gfCNCPoint5[28762] = {X 295.8044, Y 11.0396, Z -8.0000, A 0.000, B 0.000, C 0.000 }
gfCNCPoint5[28763] = {X 295.9180, Y 11.7127, Z -8.0000, A 0.000, B 0.000, C 0.000 }
gfCNCPoint5[28764] = {X 295.9354, Y 11.9495, Z -8.0000, A 0.000, B 0.000, C 0.000 }
gfCNCPoint5[28765] = {X 295.9411, Y 12.1868, Z -8.0000, A 0.000, B 0.000, C 0.000 }
gfCNCPoint5[28766] = {X 295.9409, Y 13.0237, Z -8.0000, A 0.000, B 0.000, C 0.000 }
gfCNCPoint5[28767] = {X 295.9342, Y 13.2382, Z -8.0000, A 0.000, B 0.000, C 0.000 }
gfCNCPoint5[28768] = {X 295.9180, Y 13.4521, Z -8.0000, A 0.000, B 0.000, C 0.000 }
gfCNCPoint5[28769] = {X 298.3067, Y 13.6853, Z -8.0000, A 0.000, B 0.000, C 0.000 }
gfCNCPoint5[28770] = {X 298.1362, Y 14.6931, Z -8.0000, A 0.000, B 0.000, C 0.000 }
gfCNCPoint5[28771] = {X 297.8263, Y 15.6671, Z -8.0000, A 0.000, B 0.000, C 0.000 }
gfCNCPoint5[28772] = {X 297.3830, Y 16.5881, Z -8.0000, A 0.000, B 0.000, C 0.000 }
gfCNCPoint5[28773] = {X 296.8150, Y 17.4380, Z -8.0000, A 0.000, B 0.000, C 0.000 }
gfCNCPoint5[28774] = {X 296.8153, Y 19.2365, Z -8.0000, A 0.000, B 0.000, C 0.000 }
gfCNCPoint5[28775] = {X 299.7981, Y 19.2365, Z -8.0000, A 0.000, B 0.000, C 0.000 }
gfCNCPoint5[28776] = {X 299.7982, Y 17.4377, Z -8.0000, A 0.000, B 0.000, C 0.000 }
gfCNCPoint5[28777] = {X 299.2303, Y 16.5879, Z -8.0000, A 0.000, B 0.000, C 0.000 }
gfCNCPoint5[28778] = {X 298.7871, Y 15.6670, Z -8.0000, A 0.000, B 0.000, C 0.000 }
gfCNCPoint5[28779] = {X 298.4771, Y 14.6930, Z -8.0000, A 0.000, B 0.000, C 0.000 }
gfCNCPoint5[28780] = {X 298.3067, Y 13.6853, Z -8.0000, A 0.000, B 0.000, C 0.000 }
gfCNCPoint5[28781] = {X 295.9180, Y 13.4521, Z -8.0000, A 0.000, B 0.000, C 0.000 }
gfCNCPoint5[28782] = {X 295.7561, Y 14.3091, Z -8.0000, A 0.000, B 0.000, C 0.000 }
gfCNCPoint5[28783] = {X 295.4442, Y 15.1235, Z -8.0000, A 0.000, B 0.000, C 0.000 }
gfCNCPoint5[28784] = {X 294.9923, Y 15.8694, Z -8.0000, A 0.000, B 0.000, C 0.000 }
gfCNCPoint5[28785] = {X 294.4149, Y 16.5230, Z -8.0000, A 0.000, B 0.000, C 0.000 }
gfCNCPoint5[28786] = {X 294.4149, Y 16.7686, Z -8.0000, A 0.000, B 0.000, C 0.000 }
gfCNCPoint5[28787] = {X 294.4156, Y 21.6365, Z -8.0000, A 0.000, B 0.000, C 0.000 }
gfCNCPoint5[28788] = {X 302.1980, Y 21.6365, Z -8.0000, A 0.000, B 0.000, C 0.000 }
gfCNCPoint5[28789] = {X 302.1982, Y 16.5227, Z -8.0000, A 0.000, B 0.000, C 0.000 }
gfCNCPoint5[28790] = {X 301.6209, Y 15.8692, Z -8.0000, A 0.000, B 0.000, C 0.000 }
gfCNCPoint5[28791] = {X 301.1691, Y 15.1233, Z -8.0000, A 0.000, B 0.000, C 0.000 }
gfCNCPoint5[28792] = {X 300.8573, Y 14.3090, Z -8.0000, A 0.000, B 0.000, C 0.000 }
gfCNCPoint5[28793] = {X 300.6953, Y 13.4521, Z -8.0000, A 0.000, B 0.000, C 0.000 }
gfCNCPoint5[28794] = {X 300.6791, Y 13.2371, Z -8.0000, A 0.000, B 0.000, C 0.000 }
gfCNCPoint5[28795] = {X 300.6724, Y 13.0215, Z -8.0000, A 0.000, B 0.000, C 0.000 }
gfCNCPoint5[28796] = {X 300.6723, Y 12.1868, Z -8.0000, A 0.000, B 0.000, C 0.000 }
gfCNCPoint5[28797] = {X 300.6780, Y 11.9495, Z -8.0000, A 0.000, B 0.000, C 0.000 }
gfCNCPoint5[28798] = {X 300.6953, Y 11.7127, Z -8.0000, A 0.000, B 0.000, C 0.000 }
gfCNCPoint5[28799] = {X 300.8090, Y 11.0396, Z -8.0000, A 0.000, B 0.000, C 0.000 }
gfCNCPoint5[28800] = {X 301.0155, Y 10.3890, Z -8.0000, A 0.000, B 0.000, C 0.000 }
gfCNCPoint5[28801] = {X 301.4602, Y 9.5279, Z -8.0000, A 0.000, B 0.000, C 0.000 }
gfCNCPoint5[28802] = {X 302.0663, Y 8.7718, Z -8.0000, A 0.000, B 0.000, C 0.000 }
gfCNCPoint5[28803] = {X 302.8099, Y 8.1502, Z -8.0000, A 0.000, B 0.000, C 0.000 }
gfCNCPoint5[28804] = {X 303.6616, Y 7.6879, Z -8.0000, A 0.000, B 0.000, C 0.000 }
gfCNCPoint5[28805] = {X 304.5879, Y 7.4030, Z -8.0000, A 0.000, B 0.000, C 0.000 }
gfCNCPoint5[28806] = {X 305.5523, Y 7.3068, Z -8.0000, A 0.000, B 0.000, C 0.000 }
gfCNCPoint5[28807] = {X 311.9957, Y 7.3068, Z -8.0000, A 0.000, B 0.000, C 0.000 }
gfCNCPoint5[28808] = {X 312.9478, Y 7.4006, Z -8.0000, A 0.000, B 0.000, C 0.000 }
gfCNCPoint5[28809] = {X 313.8632, Y 7.6783, Z -8.0000, A 0.000, B 0.000, C 0.000 }
gfCNCPoint5[28810] = {X 314.7069, Y 8.1292, Z -8.0000, A 0.000, B 0.000, C 0.000 }
gfCNCPoint5[28811] = {X 315.4464, Y 8.7361, Z -8.0000, A 0.000, B 0.000, C 0.000 }
gfCNCPoint5[28812] = {X 316.0533, Y 9.4756, Z -8.0000, A 0.000, B 0.000, C 0.000 }
gfCNCPoint5[28813] = {X 316.5043, Y 10.3193, Z -8.0000, A 0.000, B 0.000, C 0.000 }
gfCNCPoint5[28814] = {X 316.7820, Y 11.2348, Z -8.0000, A 0.000, B 0.000, C 0.000 }
gfCNCPoint5[28815] = {X 316.8757, Y 12.1868, Z -8.0000, A 0.000, B 0.000, C 0.000 }
gfCNCPoint5[28816] = {X 316.8755, Y 13.0237, Z -8.0000, A 0.000, B 0.000, C 0.000 }
gfCNCPoint5[28817] = {X 316.7682, Y 13.9967, Z -8.0000, A 0.000, B 0.000, C 0.000 }
gfCNCPoint5[28818] = {X 316.4689, Y 14.9287, Z -8.0000, A 0.000, B 0.000, C 0.000 }
gfCNCPoint5[28819] = {X 315.9896, Y 15.7823, Z -8.0000, A 0.000, B 0.000, C 0.000 }
gfCNCPoint5[28820] = {X 315.3495, Y 16.5229, Z -8.0000, A 0.000, B 0.000, C 0.000 }
gfCNCPoint5[28821] = {X 315.3493, Y 40.6637, Z -8.0000, A 0.000, B 0.000, C 0.000 }
gfCNCPoint5[28822] = {X 315.9899, Y 41.4051, Z -8.0000, A 0.000, B 0.000, C 0.000 }
gfCNCPoint5[28823] = {X 316.4695, Y 42.2595, Z -8.0000, A 0.000, B 0.000, C 0.000 }
gfCNCPoint5[28824] = {X 316.7687, Y 43.1925, Z -8.0000, A 0.000, B 0.000, C 0.000 }
gfCNCPoint5[28825] = {X 316.8755, Y 44.1664, Z -8.0000, A 0.000, B 0.000, C 0.000 }
gfCNCPoint5[28826] = {X 316.8757, Y 45.0000, Z -8.0000, A 0.000, B 0.000, C 0.000 }
gfCNCPoint5[28827] = {X 316.8749, Y 45.0899, Z -8.0000, A 0.000, B 0.000, C 0.000 }
gfCNCPoint5[28828] = {X 316.8724, Y 45.1799, Z -8.0000, A 0.000, B 0.000, C 0.000 }
gfCNCPoint5[28829] = {X 316.8594, Y 45.3987, Z -8.0000, A 0.000, B 0.000, C 0.000 }
gfCNCPoint5[28830] = {X 316.8366, Y 45.6167, Z -8.0000, A 0.000, B 0.000, C 0.000 }
gfCNCPoint5[28831] = {X 316.6062, Y 46.5992, Z -8.0000, A 0.000, B 0.000, C 0.000 }
gfCNCPoint5[28832] = {X 316.1787, Y 47.5134, Z -8.0000, A 0.000, B 0.000, C 0.000 }
gfCNCPoint5[28833] = {X 315.5723, Y 48.3200, Z -8.0000, A 0.000, B 0.000, C 0.000 }
gfCNCPoint5[28834] = {X 315.2205, Y 47.9934, Z -8.0000, A 0.000, B 0.000, C 0.000 }
gfCNCPoint5[28835] = {X 314.5413, Y 48.5889, Z -8.0000, A 0.000, B 0.000, C 0.000 }
gfCNCPoint5[28836] = {X 313.7548, Y 49.0331, Z -8.0000, A 0.000, B 0.000, C 0.000 }
gfCNCPoint5[28837] = {X 312.8942, Y 49.3073, Z -8.0000, A 0.000, B 0.000, C 0.000 }
gfCNCPoint5[28838] = {X 311.9957, Y 49.4000, Z -8.0000, A 0.000, B 0.000, C 0.000 }
gfCNCPoint5[28839] = {X 305.5523, Y 49.4000, Z -8.0000, A 0.000, B 0.000, C 0.000 }
gfCNCPoint5[28840] = {X 304.5732, Y 49.2897, Z -8.0000, A 0.000, B 0.000, C 0.000 }
gfCNCPoint5[28841] = {X 303.6432, Y 48.9643, Z -8.0000, A 0.000, B 0.000, C 0.000 }
gfCNCPoint5[28842] = {X 302.8089, Y 48.4401, Z -8.0000, A 0.000, B 0.000, C 0.000 }
gfCNCPoint5[28843] = {X 302.1122, Y 47.7433, Z -8.0000, A 0.000, B 0.000, C 0.000 }
gfCNCPoint5[28844] = {X 301.5880, Y 46.9091, Z -8.0000, A 0.000, B 0.000, C 0.000 }
gfCNCPoint5[28845] = {X 301.2626, Y 45.9791, Z -8.0000, A 0.000, B 0.000, C 0.000 }
gfCNCPoint5[28846] = {X 301.1523, Y 45.0000, Z -8.0000, A 0.000, B 0.000, C 0.000 }
gfCNCPoint5[28847] = {X 301.1524, Y 44.1996, Z -8.0000, A 0.000, B 0.000, C 0.000 }
gfCNCPoint5[28848] = {X 301.2693, Y 43.2561, Z -8.0000, A 0.000, B 0.000, C 0.000 }
gfCNCPoint5[28849] = {X 301.5719, Y 42.3548, Z -8.0000, A 0.000, B 0.000, C 0.000 }
gfCNCPoint5[28850] = {X 302.0480, Y 41.5318, Z -8.0000, A 0.000, B 0.000, C 0.000 }
gfCNCPoint5[28851] = {X 302.6784, Y 40.8201, Z -8.0000, A 0.000, B 0.000, C 0.000 }
gfCNCPoint5[28852] = {X 302.6784, Y 34.1143, Z -8.0000, A 0.000, B 0.000, C 0.000 }
gfCNCPoint5[28853] = {X 293.9354, Y 34.1143, Z -8.0000, A 0.000, B 0.000, C 0.000 }
gfCNCPoint5[28854] = {X 293.9349, Y 40.8654, Z -8.0000, A 0.000, B 0.000, C 0.000 }
gfCNCPoint5[28855] = {X 294.5750, Y 41.5604, Z -8.0000, A 0.000, B 0.000, C 0.000 }
gfCNCPoint5[28856] = {X 295.0555, Y 42.3739, Z -8.0000, A 0.000, B 0.000, C 0.000 }
gfCNCPoint5[28857] = {X 295.3554, Y 43.2699, Z -8.0000, A 0.000, B 0.000, C 0.000 }
gfCNCPoint5[28858] = {X 295.4611, Y 44.2088, Z -8.0000, A 0.000, B 0.000, C 0.000 }
gfCNCPoint5[28859] = {X 295.4611, Y 45.0000, Z -8.0000, A 0.000, B 0.000, C 0.000 }
gfCNCPoint5[28860] = {X 295.3508, Y 45.9791, Z -8.0000, A 0.000, B 0.000, C 0.000 }
gfCNCPoint5[28861] = {X 295.0254, Y 46.9091, Z -8.0000, A 0.000, B 0.000, C 0.000 }
gfCNCPoint5[28862] = {X 294.5012, Y 47.7434, Z -8.0000, A 0.000, B 0.000, C 0.000 }
gfCNCPoint5[28863] = {X 293.8045, Y 48.4401, Z -8.0000, A 0.000, B 0.000, C 0.000 }
gfCNCPoint5[28864] = {X 292.9702, Y 48.9643, Z -8.0000, A 0.000, B 0.000, C 0.000 }
gfCNCPoint5[28865] = {X 292.0402, Y 49.2897, Z -8.0000, A 0.000, B 0.000, C 0.000 }
gfCNCPoint5[28866] = {X 291.0611, Y 49.4000, Z -8.0000, A 0.000, B 0.000, C 0.000 }
gfCNCPoint5[28867] = {X 284.6177, Y 49.4000, Z -8.0000, A 0.000, B 0.000, C 0.000 }
gfCNCPoint5[28868] = {X 283.6386, Y 49.2897, Z -8.0000, A 0.000, B 0.000, C 0.000 }
gfCNCPoint5[28869] = {X 282.7086, Y 48.9643, Z -8.0000, A 0.000, B 0.000, C 0.000 }
gfCNCPoint5[28870] = {X 281.8743, Y 48.4401, Z -8.0000, A 0.000, B 0.000, C 0.000 }
gfCNCPoint5[28871] = {X 281.1776, Y 47.7433, Z -8.0000, A 0.000, B 0.000, C 0.000 }
gfCNCPoint5[28872] = {X 280.6534, Y 46.9091, Z -8.0000, A 0.000, B 0.000, C 0.000 }
gfCNCPoint5[28873] = {X 280.3280, Y 45.9791, Z -8.0000, A 0.000, B 0.000, C 0.000 }
gfCNCPoint5[28874] = {X 280.2177, Y 45.0000, Z -8.0000, A 0.000, B 0.000, C 0.000 }
gfCNCPoint5[28875] = {X 280.2177, Y 44.2072, Z -8.0000, A 0.000, B 0.000, C 0.000 }
gfCNCPoint5[28876] = {X 280.3216, Y 43.2699, Z -8.0000, A 0.000, B 0.000, C 0.000 }
gfCNCPoint5[28877] = {X 280.6210, Y 42.3756, Z -8.0000, A 0.000, B 0.000, C 0.000 }
gfCNCPoint5[28878] = {X 281.1024, Y 41.5647, Z -8.0000, A 0.000, B 0.000, C 0.000 }
gfCNCPoint5[28879] = {X 281.7441, Y 40.8737, Z -8.0000, A 0.000, B 0.000, C 0.000 }
gfCNCPoint5[28880] = {X 281.7443, Y 16.3102, Z -8.0000, A 0.000, B 0.000, C 0.000 }
gfCNCPoint5[28881] = {X 281.1000, Y 15.6212, Z -8.0000, A 0.000, B 0.000, C 0.000 }
gfCNCPoint5[28882] = {X 280.6175, Y 14.8106, Z -8.0000, A 0.000, B 0.000, C 0.000 }
gfCNCPoint5[28883] = {X 280.3188, Y 13.9159, Z -8.0000, A 0.000, B 0.000, C 0.000 }
gfCNCPoint5[28884] = {X 280.2177, Y 12.9780, Z -8.0000, A 0.000, B 0.000, C 0.000 }
gfCNCPoint5[28885] = {X 280.2177, Y 12.1868, Z -8.0000, A 0.000, B 0.000, C 0.000 }
gfCNCPoint5[28886] = {X 280.3280, Y 11.2077, Z -8.0000, A 0.000, B 0.000, C 0.000 }
gfCNCPoint5[28887] = {X 280.6534, Y 10.2777, Z -8.0000, A 0.000, B 0.000, C 0.000 }
gfCNCPoint5[28888] = {X 281.1776, Y 9.4435, Z -8.0000, A 0.000, B 0.000, C 0.000 }
gfCNCPoint5[28889] = {X 281.8743, Y 8.7468, Z -8.0000, A 0.000, B 0.000, C 0.000 }
gfCNCPoint5[28890] = {X 282.7086, Y 8.2226, Z -8.0000, A 0.000, B 0.000, C 0.000 }
gfCNCPoint5[28891] = {X 283.6386, Y 7.8971, Z -8.0000, A 0.000, B 0.000, C 0.000 }
gfCNCPoint5[28892] = {X 284.6177, Y 7.7868, Z -8.0000, A 0.000, B 0.000, C 0.000 }
gfCNCPoint5[28893] = {X 291.0611, Y 7.7868, Z -8.0000, A 0.000, B 0.000, C 0.000 }
gfCNCPoint5[28894] = {X 292.0402, Y 7.8971, Z -8.0000, A 0.000, B 0.000, C 0.000 }
gfCNCPoint5[28895] = {X 292.9702, Y 8.2226, Z -8.0000, A 0.000, B 0.000, C 0.000 }
gfCNCPoint5[28896] = {X 293.8045, Y 8.7468, Z -8.0000, A 0.000, B 0.000, C 0.000 }
gfCNCPoint5[28897] = {X 294.5012, Y 9.4435, Z -8.0000, A 0.000, B 0.000, C 0.000 }
gfCNCPoint5[28898] = {X 295.0254, Y 10.2777, Z -8.0000, A 0.000, B 0.000, C 0.000 }
gfCNCPoint5[28899] = {X 295.3508, Y 11.2077, Z -8.0000, A 0.000, B 0.000, C 0.000 }
gfCNCPoint5[28900] = {X 295.4611, Y 12.1868, Z -8.0000, A 0.000, B 0.000, C 0.000 }
gfCNCPoint5[28901] = {X 295.4609, Y 13.0233, Z -8.0000, A 0.000, B 0.000, C 0.000 }
gfCNCPoint5[28902] = {X 295.3527, Y 13.9490, Z -8.0000, A 0.000, B 0.000, C 0.000 }
gfCNCPoint5[28903] = {X 295.0519, Y 14.8311, Z -8.0000, A 0.000, B 0.000, C 0.000 }
gfCNCPoint5[28904] = {X 294.5721, Y 15.6300, Z -8.0000, A 0.000, B 0.000, C 0.000 }
gfCNCPoint5[28905] = {X 293.9348, Y 16.3100, Z -8.0000, A 0.000, B 0.000, C 0.000 }
gfCNCPoint5[28906] = {X 293.9349, Y 16.7687, Z -8.0000, A 0.000, B 0.000, C 0.000 }
gfCNCPoint5[28907] = {X 293.9356, Y 22.1165, Z -8.0000, A 0.000, B 0.000, C 0.000 }
gfCNCPoint5[28908] = {X 302.6780, Y 22.1165, Z -8.0000, A 0.000, B 0.000, C 0.000 }
gfCNCPoint5[28909] = {X 302.6782, Y 16.3097, Z -8.0000, A 0.000, B 0.000, C 0.000 }
gfCNCPoint5[28910] = {X 302.0342, Y 15.6207, Z -8.0000, A 0.000, B 0.000, C 0.000 }
gfCNCPoint5[28911] = {X 301.5519, Y 14.8102, Z -8.0000, A 0.000, B 0.000, C 0.000 }
gfCNCPoint5[28912] = {X 301.2533, Y 13.9156, Z -8.0000, A 0.000, B 0.000, C 0.000 }
gfCNCPoint5[28913] = {X 301.1523, Y 12.9780, Z -8.0000, A 0.000, B 0.000, C 0.000 }
gfCNCPoint5[28914] = {X 301.1523, Y 12.1868, Z -8.0000, A 0.000, B 0.000, C 0.000 }
gfCNCPoint5[28915] = {X 301.2626, Y 11.2077, Z -8.0000, A 0.000, B 0.000, C 0.000 }
gfCNCPoint5[28916] = {X 301.5880, Y 10.2777, Z -8.0000, A 0.000, B 0.000, C 0.000 }
gfCNCPoint5[28917] = {X 302.1122, Y 9.4435, Z -8.0000, A 0.000, B 0.000, C 0.000 }
gfCNCPoint5[28918] = {X 302.8089, Y 8.7468, Z -8.0000, A 0.000, B 0.000, C 0.000 }
gfCNCPoint5[28919] = {X 303.6432, Y 8.2226, Z -8.0000, A 0.000, B 0.000, C 0.000 }
gfCNCPoint5[28920] = {X 304.5732, Y 7.8971, Z -8.0000, A 0.000, B 0.000, C 0.000 }
gfCNCPoint5[28921] = {X 305.5523, Y 7.7868, Z -8.0000, A 0.000, B 0.000, C 0.000 }
gfCNCPoint5[28922] = {X 311.9957, Y 7.7868, Z -8.0000, A 0.000, B 0.000, C 0.000 }
gfCNCPoint5[28923] = {X 312.9748, Y 7.8971, Z -8.0000, A 0.000, B 0.000, C 0.000 }
gfCNCPoint5[28924] = {X 313.9048, Y 8.2226, Z -8.0000, A 0.000, B 0.000, C 0.000 }
gfCNCPoint5[28925] = {X 314.7391, Y 8.7468, Z -8.0000, A 0.000, B 0.000, C 0.000 }
gfCNCPoint5[28926] = {X 315.4358, Y 9.4435, Z -8.0000, A 0.000, B 0.000, C 0.000 }
gfCNCPoint5[28927] = {X 315.9600, Y 10.2777, Z -8.0000, A 0.000, B 0.000, C 0.000 }
gfCNCPoint5[28928] = {X 316.2854, Y 11.2077, Z -8.0000, A 0.000, B 0.000, C 0.000 }
gfCNCPoint5[28929] = {X 316.3957, Y 12.1868, Z -8.0000, A 0.000, B 0.000, C 0.000 }
gfCNCPoint5[28930] = {X 316.3955, Y 13.0233, Z -8.0000, A 0.000, B 0.000, C 0.000 }
gfCNCPoint5[28931] = {X 316.2873, Y 13.9489, Z -8.0000, A 0.000, B 0.000, C 0.000 }
gfCNCPoint5[28932] = {X 315.9865, Y 14.8310, Z -8.0000, A 0.000, B 0.000, C 0.000 }
gfCNCPoint5[28933] = {X 315.5068, Y 15.6299, Z -8.0000, A 0.000, B 0.000, C 0.000 }
gfCNCPoint5[28934] = {X 314.8695, Y 16.3099, Z -8.0000, A 0.000, B 0.000, C 0.000 }
gfCNCPoint5[28935] = {X 314.8693, Y 40.8767, Z -8.0000, A 0.000, B 0.000, C 0.000 }
gfCNCPoint5[28936] = {X 315.5135, Y 41.5658, Z -8.0000, A 0.000, B 0.000, C 0.000 }
gfCNCPoint5[28937] = {X 315.9960, Y 42.3763, Z -8.0000, A 0.000, B 0.000, C 0.000 }
gfCNCPoint5[28938] = {X 316.2946, Y 43.2710, Z -8.0000, A 0.000, B 0.000, C 0.000 }
gfCNCPoint5[28939] = {X 316.3957, Y 44.2089, Z -8.0000, A 0.000, B 0.000, C 0.000 }
gfCNCPoint5[28940] = {X 316.3957, Y 45.0000, Z -8.0000, A 0.000, B 0.000, C 0.000 }
gfCNCPoint5[28941] = {X 316.3190, Y 45.8182, Z -8.0000, A 0.000, B 0.000, C 0.000 }
gfCNCPoint5[28942] = {X 316.0914, Y 46.6079, Z -8.0000, A 0.000, B 0.000, C 0.000 }
gfCNCPoint5[28943] = {X 315.7209, Y 47.3415, Z -8.0000, A 0.000, B 0.000, C 0.000 }
gfCNCPoint5[28944] = {X 315.2205, Y 47.9934, Z -8.0000, A 0.000, B 0.000, C 0.000 }
gfCNCPoint5[28945] = {X 315.5723, Y 48.3200, Z -8.0000, A 0.000, B 0.000, C 0.000 }
gfCNCPoint5[28946] = {X 324.3107, Y 48.3200, Z -8.0000, A 0.000, B 0.000, C 0.000 }
gfCNCPoint5[28947] = {X 325.5555, Y 48.4004, Z -8.0000, A 0.000, B 0.000, C 0.000 }
gfCNCPoint5[28948] = {X 326.7797, Y 48.6402, Z -8.0000, A 0.000, B 0.000, C 0.000 }
gfCNCPoint5[28949] = {X 325.5882, Y 48.0963, Z -8.0000, A 0.000, B 0.000, C 0.000 }
gfCNCPoint5[28950] = {X 324.4810, Y 47.3966, Z -8.0000, A 0.000, B 0.000, C 0.000 }
gfCNCPoint5[28951] = {X 323.4784, Y 46.5538, Z -8.0000, A 0.000, B 0.000, C 0.000 }
gfCNCPoint5[28952] = {X 322.8382, Y 45.9295, Z -8.0000, A 0.000, B 0.000, C 0.000 }
gfCNCPoint5[28953] = {X 322.2180, Y 45.2650, Z -8.0000, A 0.000, B 0.000, C 0.000 }
gfCNCPoint5[28954] = {X 321.6628, Y 44.5452, Z -8.0000, A 0.000, B 0.000, C 0.000 }
gfCNCPoint5[28955] = {X 323.6300, Y 43.1703, Z -8.0000, A 0.000, B 0.000, C 0.000 }
gfCNCPoint5[28956] = {X 323.0063, Y 42.0918, Z -8.0000, A 0.000, B 0.000, C 0.000 }
gfCNCPoint5[28957] = {X 322.5757, Y 40.9227, Z -8.0000, A 0.000, B 0.000, C 0.000 }
gfCNCPoint5[28958] = {X 322.3506, Y 39.6973, Z -8.0000, A 0.000, B 0.000, C 0.000 }
gfCNCPoint5[28959] = {X 322.3379, Y 38.4514, Z -8.0000, A 0.000, B 0.000, C 0.000 }
gfCNCPoint5[28960] = {X 322.5377, Y 37.2217, Z -8.0000, A 0.000, B 0.000, C 0.000 }
gfCNCPoint5[28961] = {X 322.9443, Y 36.0440, Z -8.0000, A 0.000, B 0.000, C 0.000 }
gfCNCPoint5[28962] = {X 323.5458, Y 34.9529, Z -8.0000, A 0.000, B 0.000, C 0.000 }
gfCNCPoint5[28963] = {X 327.7840, Y 28.6158, Z -8.0000, A 0.000, B 0.000, C 0.000 }
gfCNCPoint5[28964] = {X 328.5200, Y 27.6906, Z -8.0000, A 0.000, B 0.000, C 0.000 }
gfCNCPoint5[28965] = {X 329.3960, Y 26.8968, Z -8.0000, A 0.000, B 0.000, C 0.000 }
gfCNCPoint5[28966] = {X 330.3889, Y 26.2552, Z -8.0000, A 0.000, B 0.000, C 0.000 }
gfCNCPoint5[28967] = {X 331.5063, Y 25.7713, Z -8.0000, A 0.000, B 0.000, C 0.000 }
gfCNCPoint5[28968] = {X 332.6887, Y 25.4804, Z -8.0000, A 0.000, B 0.000, C 0.000 }
gfCNCPoint5[28969] = {X 333.9031, Y 25.3907, Z -8.0000, A 0.000, B 0.000, C 0.000 }
gfCNCPoint5[28970] = {X 335.1154, Y 25.5046, Z -8.0000, A 0.000, B 0.000, C 0.000 }
gfCNCPoint5[28971] = {X 336.2918, Y 25.8191, Z -8.0000, A 0.000, B 0.000, C 0.000 }
gfCNCPoint5[28972] = {X 337.3993, Y 26.3252, Z -8.0000, A 0.000, B 0.000, C 0.000 }
gfCNCPoint5[28973] = {X 338.1754, Y 26.8291, Z -8.0000, A 0.000, B 0.000, C 0.000 }
gfCNCPoint5[28974] = {X 338.8812, Y 27.4274, Z -8.0000, A 0.000, B 0.000, C 0.000 }
gfCNCPoint5[28975] = {X 339.5028, Y 28.0267, Z -8.0000, A 0.000, B 0.000, C 0.000 }
gfCNCPoint5[28976] = {X 340.3317, Y 28.9981, Z -8.0000, A 0.000, B 0.000, C 0.000 }
gfCNCPoint5[28977] = {X 340.9781, Y 30.0993, Z -8.0000, A 0.000, B 0.000, C 0.000 }
gfCNCPoint5[28978] = {X 341.4222, Y 31.2965, Z -8.0000, A 0.000, B 0.000, C 0.000 }
gfCNCPoint5[28979] = {X 341.6502, Y 32.5529, Z -8.0000, A 0.000, B 0.000, C 0.000 }
gfCNCPoint5[28980] = {X 342.6387, Y 33.2799, Z -8.0000, A 0.000, B 0.000, C 0.000 }
gfCNCPoint5[28981] = {X 343.7299, Y 33.8413, Z -8.0000, A 0.000, B 0.000, C 0.000 }
gfCNCPoint5[28982] = {X 344.8962, Y 34.2227, Z -8.0000, A 0.000, B 0.000, C 0.000 }
gfCNCPoint5[28983] = {X 346.1081, Y 34.4147, Z -8.0000, A 0.000, B 0.000, C 0.000 }
gfCNCPoint5[28984] = {X 347.3352, Y 34.4123, Z -8.0000, A 0.000, B 0.000, C 0.000 }
gfCNCPoint5[28985] = {X 348.3044, Y 34.2866, Z -8.0000, A 0.000, B 0.000, C 0.000 }
gfCNCPoint5[28986] = {X 349.2397, Y 34.0036, Z -8.0000, A 0.000, B 0.000, C 0.000 }
gfCNCPoint5[28987] = {X 350.1160, Y 33.5708, Z -8.0000, A 0.000, B 0.000, C 0.000 }
gfCNCPoint5[28988] = {X 350.9093, Y 33.0001, Z -8.0000, A 0.000, B 0.000, C 0.000 }
gfCNCPoint5[28989] = {X 351.7850, Y 32.1491, Z -8.0000, A 0.000, B 0.000, C 0.000 }
gfCNCPoint5[28990] = {X 352.5431, Y 31.1918, Z -8.0000, A 0.000, B 0.000, C 0.000 }
gfCNCPoint5[28991] = {X 353.1707, Y 30.1444, Z -8.0000, A 0.000, B 0.000, C 0.000 }
gfCNCPoint5[28992] = {X 353.6573, Y 29.0244, Z -8.0000, A 0.000, B 0.000, C 0.000 }
gfCNCPoint5[28993] = {X 353.9945, Y 27.8508, Z -8.0000, A 0.000, B 0.000, C 0.000 }
gfCNCPoint5[28994] = {X 354.2220, Y 26.4400, Z -8.0000, A 0.000, B 0.000, C 0.000 }
gfCNCPoint5[28995] = {X 354.3140, Y 25.0140, Z -8.0000, A 0.000, B 0.000, C 0.000 }
gfCNCPoint5[28996] = {X 354.2698, Y 23.5857, Z -8.0000, A 0.000, B 0.000, C 0.000 }
gfCNCPoint5[28997] = {X 354.0897, Y 22.1681, Z -8.0000, A 0.000, B 0.000, C 0.000 }
gfCNCPoint5[28998] = {X 353.8250, Y 21.0254, Z -8.0000, A 0.000, B 0.000, C 0.000 }
gfCNCPoint5[28999] = {X 353.4119, Y 19.9275, Z -8.0000, A 0.000, B 0.000, C 0.000 }
gfCNCPoint5[29000] = {X 352.8576, Y 18.8937, Z -8.0000, A 0.000, B 0.000, C 0.000 }
gfCNCPoint5[29001] = {X 352.1718, Y 17.9421, Z -8.0000, A 0.000, B 0.000, C 0.000 }
gfCNCPoint5[29002] = {X 351.4219, Y 17.1690, Z -8.0000, A 0.000, B 0.000, C 0.000 }
gfCNCPoint5[29003] = {X 350.5492, Y 16.5376, Z -8.0000, A 0.000, B 0.000, C 0.000 }
gfCNCPoint5[29004] = {X 349.5804, Y 16.0671, Z -8.0000, A 0.000, B 0.000, C 0.000 }
gfCNCPoint5[29005] = {X 348.5446, Y 15.7717, Z -8.0000, A 0.000, B 0.000, C 0.000 }
gfCNCPoint5[29006] = {X 347.1584, Y 15.5996, Z -8.0000, A 0.000, B 0.000, C 0.000 }
gfCNCPoint5[29007] = {X 345.7616, Y 15.6148, Z -8.0000, A 0.000, B 0.000, C 0.000 }
gfCNCPoint5[29008] = {X 344.3794, Y 15.8170, Z -8.0000, A 0.000, B 0.000, C 0.000 }
gfCNCPoint5[29009] = {X 343.0368, Y 16.2026, Z -8.0000, A 0.000, B 0.000, C 0.000 }
gfCNCPoint5[29010] = {X 341.7580, Y 16.7646, Z -8.0000, A 0.000, B 0.000, C 0.000 }
gfCNCPoint5[29011] = {X 341.4304, Y 17.8590, Z -8.0000, A 0.000, B 0.000, C 0.000 }
gfCNCPoint5[29012] = {X 340.9357, Y 18.8888, Z -8.0000, A 0.000, B 0.000, C 0.000 }
gfCNCPoint5[29013] = {X 340.2859, Y 19.8284, Z -8.0000, A 0.000, B 0.000, C 0.000 }
gfCNCPoint5[29014] = {X 345.8684, Y 24.3755, Z -8.0000, A 0.000, B 0.000, C 0.000 }
gfCNCPoint5[29015] = {X 346.4660, Y 25.2106, Z -8.0000, A 0.000, B 0.000, C 0.000 }
gfCNCPoint5[29016] = {X 347.0029, Y 26.0860, Z -8.0000, A 0.000, B 0.000, C 0.000 }
gfCNCPoint5[29017] = {X 347.1049, Y 25.1804, Z -8.0000, A 0.000, B 0.000, C 0.000 }
gfCNCPoint5[29018] = {X 347.1005, Y 24.2691, Z -8.0000, A 0.000, B 0.000, C 0.000 }
gfCNCPoint5[29019] = {X 346.9895, Y 23.3646, Z -8.0000, A 0.000, B 0.000, C 0.000 }
gfCNCPoint5[29020] = {X 346.9483, Y 23.1618, Z -8.0000, A 0.000, B 0.000, C 0.000 }
gfCNCPoint5[29021] = {X 346.8824, Y 22.9657, Z -8.0000, A 0.000, B 0.000, C 0.000 }
gfCNCPoint5[29022] = {X 346.3965, Y 23.6858, Z -8.0000, A 0.000, B 0.000, C 0.000 }
gfCNCPoint5[29023] = {X 345.8684, Y 24.3755, Z -8.0000, A 0.000, B 0.000, C 0.000 }
gfCNCPoint5[29024] = {X 344.0076, Y 22.8598, Z -8.0000, A 0.000, B 0.000, C 0.000 }
gfCNCPoint5[29025] = {X 343.3277, Y 23.6257, Z -8.0000, A 0.000, B 0.000, C 0.000 }
gfCNCPoint5[29026] = {X 342.5854, Y 24.3313, Z -8.0000, A 0.000, B 0.000, C 0.000 }
gfCNCPoint5[29027] = {X 343.4620, Y 25.2275, Z -8.0000, A 0.000, B 0.000, C 0.000 }
gfCNCPoint5[29028] = {X 344.2409, Y 26.2098, Z -8.0000, A 0.000, B 0.000, C 0.000 }
gfCNCPoint5[29029] = {X 344.9138, Y 27.2675, Z -8.0000, A 0.000, B 0.000, C 0.000 }
gfCNCPoint5[29030] = {X 345.4656, Y 28.3710, Z -8.0000, A 0.000, B 0.000, C 0.000 }
gfCNCPoint5[29031] = {X 345.9019, Y 29.5251, Z -8.0000, A 0.000, B 0.000, C 0.000 }
gfCNCPoint5[29032] = {X 346.4628, Y 29.6282, Z -8.0000, A 0.000, B 0.000, C 0.000 }
gfCNCPoint5[29033] = {X 347.0330, Y 29.6206, Z -8.0000, A 0.000, B 0.000, C 0.000 }
gfCNCPoint5[29034] = {X 347.4389, Y 29.5545, Z -8.0000, A 0.000, B 0.000, C 0.000 }
gfCNCPoint5[29035] = {X 347.7946, Y 29.3479, Z -8.0000, A 0.000, B 0.000, C 0.000 }
gfCNCPoint5[29036] = {X 348.4743, Y 28.6286, Z -8.0000, A 0.000, B 0.000, C 0.000 }
gfCNCPoint5[29037] = {X 348.9844, Y 27.7806, Z -8.0000, A 0.000, B 0.000, C 0.000 }
gfCNCPoint5[29038] = {X 349.3014, Y 26.8431, Z -8.0000, A 0.000, B 0.000, C 0.000 }
gfCNCPoint5[29039] = {X 349.3362, Y 26.6688, Z -8.0000, A 0.000, B 0.000, C 0.000 }
gfCNCPoint5[29040] = {X 349.3680, Y 26.4938, Z -8.0000, A 0.000, B 0.000, C 0.000 }
gfCNCPoint5[29041] = {X 349.5008, Y 25.3209, Z -8.0000, A 0.000, B 0.000, C 0.000 }
gfCNCPoint5[29042] = {X 349.4971, Y 24.1405, Z -8.0000, A 0.000, B 0.000, C 0.000 }
gfCNCPoint5[29043] = {X 349.3568, Y 22.9684, Z -8.0000, A 0.000, B 0.000, C 0.000 }
gfCNCPoint5[29044] = {X 349.1791, Y 22.2566, Z -8.0000, A 0.000, B 0.000, C 0.000 }
gfCNCPoint5[29045] = {X 348.8767, Y 21.5882, Z -8.0000, A 0.000, B 0.000, C 0.000 }
gfCNCPoint5[29046] = {X 348.4593, Y 20.9848, Z -8.0000, A 0.000, B 0.000, C 0.000 }
gfCNCPoint5[29047] = {X 348.0918, Y 20.6609, Z -8.0000, A 0.000, B 0.000, C 0.000 }
gfCNCPoint5[29048] = {X 347.6348, Y 20.4847, Z -8.0000, A 0.000, B 0.000, C 0.000 }
gfCNCPoint5[29049] = {X 346.5774, Y 20.3831, Z -8.0000, A 0.000, B 0.000, C 0.000 }
gfCNCPoint5[29050] = {X 345.5199, Y 20.4829, Z -8.0000, A 0.000, B 0.000, C 0.000 }
gfCNCPoint5[29051] = {X 344.8333, Y 21.7156, Z -8.0000, A 0.000, B 0.000, C 0.000 }
gfCNCPoint5[29052] = {X 344.0076, Y 22.8598, Z -8.0000, A 0.000, B 0.000, C 0.000 }
gfCNCPoint5[29053] = {X 342.1467, Y 21.3441, Z -8.0000, A 0.000, B 0.000, C 0.000 }
gfCNCPoint5[29054] = {X 341.6020, Y 21.9578, Z -8.0000, A 0.000, B 0.000, C 0.000 }
gfCNCPoint5[29055] = {X 341.0072, Y 22.5232, Z -8.0000, A 0.000, B 0.000, C 0.000 }
gfCNCPoint5[29056] = {X 340.7216, Y 22.7630, Z -8.0000, A 0.000, B 0.000, C 0.000 }
gfCNCPoint5[29057] = {X 340.4270, Y 22.9916, Z -8.0000, A 0.000, B 0.000, C 0.000 }
gfCNCPoint5[29058] = {X 339.6616, Y 23.5549, Z -8.0000, A 0.000, B 0.000, C 0.000 }
gfCNCPoint5[29059] = {X 339.1300, Y 23.9121, Z -8.0000, A 0.000, B 0.000, C 0.000 }
gfCNCPoint5[29060] = {X 338.5759, Y 24.2333, Z -8.0000, A 0.000, B 0.000, C 0.000 }
gfCNCPoint5[29061] = {X 339.6077, Y 24.9034, Z -8.0000, A 0.000, B 0.000, C 0.000 }
gfCNCPoint5[29062] = {X 340.5463, Y 25.6990, Z -8.0000, A 0.000, B 0.000, C 0.000 }
gfCNCPoint5[29063] = {X 341.1848, Y 26.3147, Z -8.0000, A 0.000, B 0.000, C 0.000 }
gfCNCPoint5[29064] = {X 342.1205, Y 27.3794, Z -8.0000, A 0.000, B 0.000, C 0.000 }
gfCNCPoint5[29065] = {X 342.8906, Y 28.5694, Z -8.0000, A 0.000, B 0.000, C 0.000 }
gfCNCPoint5[29066] = {X 343.4787, Y 29.8590, Z -8.0000, A 0.000, B 0.000, C 0.000 }
gfCNCPoint5[29067] = {X 343.8721, Y 31.2207, Z -8.0000, A 0.000, B 0.000, C 0.000 }
gfCNCPoint5[29068] = {X 344.6396, Y 31.6203, Z -8.0000, A 0.000, B 0.000, C 0.000 }
gfCNCPoint5[29069] = {X 345.4616, Y 31.8904, Z -8.0000, A 0.000, B 0.000, C 0.000 }
gfCNCPoint5[29070] = {X 346.3165, Y 32.0237, Z -8.0000, A 0.000, B 0.000, C 0.000 }
gfCNCPoint5[29071] = {X 347.1817, Y 32.0168, Z -8.0000, A 0.000, B 0.000, C 0.000 }
gfCNCPoint5[29072] = {X 347.9625, Y 31.9015, Z -8.0000, A 0.000, B 0.000, C 0.000 }
gfCNCPoint5[29073] = {X 348.6981, Y 31.6158, Z -8.0000, A 0.000, B 0.000, C 0.000 }
gfCNCPoint5[29074] = {X 349.3520, Y 31.1739, Z -8.0000, A 0.000, B 0.000, C 0.000 }
gfCNCPoint5[29075] = {X 350.1526, Y 30.3706, Z -8.0000, A 0.000, B 0.000, C 0.000 }
gfCNCPoint5[29076] = {X 350.8130, Y 29.4485, Z -8.0000, A 0.000, B 0.000, C 0.000 }
gfCNCPoint5[29077] = {X 351.3158, Y 28.4318, Z -8.0000, A 0.000, B 0.000, C 0.000 }
gfCNCPoint5[29078] = {X 351.6479, Y 27.3474, Z -8.0000, A 0.000, B 0.000, C 0.000 }
gfCNCPoint5[29079] = {X 351.8764, Y 25.7621, Z -8.0000, A 0.000, B 0.000, C 0.000 }
gfCNCPoint5[29080] = {X 351.9017, Y 24.1606, Z -8.0000, A 0.000, B 0.000, C 0.000 }
gfCNCPoint5[29081] = {X 351.7234, Y 22.5689, Z -8.0000, A 0.000, B 0.000, C 0.000 }
gfCNCPoint5[29082] = {X 351.4415, Y 21.4556, Z -8.0000, A 0.000, B 0.000, C 0.000 }
gfCNCPoint5[29083] = {X 350.9674, Y 20.4097, Z -8.0000, A 0.000, B 0.000, C 0.000 }
gfCNCPoint5[29084] = {X 350.3159, Y 19.4639, Z -8.0000, A 0.000, B 0.000, C 0.000 }
gfCNCPoint5[29085] = {X 349.6854, Y 18.8481, Z -8.0000, A 0.000, B 0.000, C 0.000 }
gfCNCPoint5[29086] = {X 348.9297, Y 18.3948, Z -8.0000, A 0.000, B 0.000, C 0.000 }
gfCNCPoint5[29087] = {X 348.0897, Y 18.1282, Z -8.0000, A 0.000, B 0.000, C 0.000 }
gfCNCPoint5[29088] = {X 346.9971, Y 17.9943, Z -8.0000, A 0.000, B 0.000, C 0.000 }
gfCNCPoint5[29089] = {X 345.8964, Y 18.0117, Z -8.0000, A 0.000, B 0.000, C 0.000 }
gfCNCPoint5[29090] = {X 344.8086, Y 18.1800, Z -8.0000, A 0.000, B 0.000, C 0.000 }
gfCNCPoint5[29091] = {X 343.7541, Y 18.4960, Z -8.0000, A 0.000, B 0.000, C 0.000 }
gfCNCPoint5[29092] = {X 343.3271, Y 19.5041, Z -8.0000, A 0.000, B 0.000, C 0.000 }
gfCNCPoint5[29093] = {X 342.7890, Y 20.4575, Z -8.0000, A 0.000, B 0.000, C 0.000 }
gfCNCPoint5[29094] = {X 342.1467, Y 21.3441, Z -8.0000, A 0.000, B 0.000, C 0.000 }
gfCNCPoint5[29095] = {X 340.2859, Y 19.8284, Z -8.0000, A 0.000, B 0.000, C 0.000 }
gfCNCPoint5[29096] = {X 339.6798, Y 20.4856, Z -8.0000, A 0.000, B 0.000, C 0.000 }
gfCNCPoint5[29097] = {X 338.9976, Y 21.0636, Z -8.0000, A 0.000, B 0.000, C 0.000 }
gfCNCPoint5[29098] = {X 338.2497, Y 21.6140, Z -8.0000, A 0.000, B 0.000, C 0.000 }
gfCNCPoint5[29099] = {X 337.8538, Y 21.8795, Z -8.0000, A 0.000, B 0.000, C 0.000 }
gfCNCPoint5[29100] = {X 337.4413, Y 22.1185, Z -8.0000, A 0.000, B 0.000, C 0.000 }
gfCNCPoint5[29101] = {X 336.3239, Y 22.6023, Z -8.0000, A 0.000, B 0.000, C 0.000 }
gfCNCPoint5[29102] = {X 335.1415, Y 22.8932, Z -8.0000, A 0.000, B 0.000, C 0.000 }
gfCNCPoint5[29103] = {X 333.9271, Y 22.9829, Z -8.0000, A 0.000, B 0.000, C 0.000 }
gfCNCPoint5[29104] = {X 332.7148, Y 22.8690, Z -8.0000, A 0.000, B 0.000, C 0.000 }
gfCNCPoint5[29105] = {X 331.5384, Y 22.5546, Z -8.0000, A 0.000, B 0.000, C 0.000 }
gfCNCPoint5[29106] = {X 330.4309, Y 22.0485, Z -8.0000, A 0.000, B 0.000, C 0.000 }
gfCNCPoint5[29107] = {X 329.5144, Y 21.4374, Z -8.0000, A 0.000, B 0.000, C 0.000 }
gfCNCPoint5[29108] = {X 328.7005, Y 20.6950, Z -8.0000, A 0.000, B 0.000, C 0.000 }
gfCNCPoint5[29109] = {X 328.0081, Y 19.8382, Z -8.0000, A 0.000, B 0.000, C 0.000 }
gfCNCPoint5[29110] = {X 327.4528, Y 18.8869, Z -8.0000, A 0.000, B 0.000, C 0.000 }
gfCNCPoint5[29111] = {X 323.9321, Y 11.6443, Z -8.0000, A 0.000, B 0.000, C 0.000 }
gfCNCPoint5[29112] = {X 323.5337, Y 10.6421, Z -8.0000, A 0.000, B 0.000, C 0.000 }
gfCNCPoint5[29113] = {X 323.2878, Y 9.5921, Z -8.0000, A 0.000, B 0.000, C 0.000 }
gfCNCPoint5[29114] = {X 323.1997, Y 8.5173, Z -8.0000, A 0.000, B 0.000, C 0.000 }
gfCNCPoint5[29115] = {X 323.2713, Y 7.4412, Z -8.0000, A 0.000, B 0.000, C 0.000 }
gfCNCPoint5[29116] = {X 323.4720, Y 6.4883, Z -8.0000, A 0.000, B 0.000, C 0.000 }
gfCNCPoint5[29117] = {X 323.7980, Y 5.5707, Z -8.0000, A 0.000, B 0.000, C 0.000 }
gfCNCPoint5[29118] = {X 324.2436, Y 4.7048, Z -8.0000, A 0.000, B 0.000, C 0.000 }
gfCNCPoint5[29119] = {X 168.0207, Y 4.7048, Z -8.0000, A 0.000, B 0.000, C 0.000 }
gfCNCPoint5[29120] = {X 168.0207, Y 9.5048, Z -8.0000, A 0.000, B 0.000, C 0.000 }
gfCNCPoint5[29121] = {X 166.5360, Y 9.5048, Z -8.0000, A 0.000, B 0.000, C 0.000 }
gfCNCPoint5[29122] = {X 166.5855, Y 9.9931, Z -8.0000, A 0.000, B 0.000, C 0.000 }
gfCNCPoint5[29123] = {X 166.6021, Y 10.4835, Z -8.0000, A 0.000, B 0.000, C 0.000 }
gfCNCPoint5[29124] = {X 166.6021, Y 13.0969, Z -8.0000, A 0.000, B 0.000, C 0.000 }
gfCNCPoint5[29125] = {X 166.8569, Y 11.8209, Z -8.0000, A 0.000, B 0.000, C 0.000 }
gfCNCPoint5[29126] = {X 167.3349, Y 10.6107, Z -8.0000, A 0.000, B 0.000, C 0.000 }
gfCNCPoint5[29127] = {X 168.0207, Y 9.5048, Z -8.0000, A 0.000, B 0.000, C 0.000 }
gfCNCPoint5[29128] = {X 168.0207, Y 7.1048, Z -8.0000, A 0.000, B 0.000, C 0.000 }
gfCNCPoint5[29129] = {X 162.8433, Y 7.1048, Z -8.0000, A 0.000, B 0.000, C 0.000 }
gfCNCPoint5[29130] = {X 163.4702, Y 7.9130, Z -8.0000, A 0.000, B 0.000, C 0.000 }
gfCNCPoint5[29131] = {X 163.9148, Y 8.8340, Z -8.0000, A 0.000, B 0.000, C 0.000 }
gfCNCPoint5[29132] = {X 164.1578, Y 9.8275, Z -8.0000, A 0.000, B 0.000, C 0.000 }
gfCNCPoint5[29133] = {X 164.1910, Y 10.1547, Z -8.0000, A 0.000, B 0.000, C 0.000 }
gfCNCPoint5[29134] = {X 164.2021, Y 10.4835, Z -8.0000, A 0.000, B 0.000, C 0.000 }
gfCNCPoint5[29135] = {X 164.2021, Y 17.4615, Z -8.0000, A 0.000, B 0.000, C 0.000 }
gfCNCPoint5[29136] = {X 164.1140, Y 18.3847, Z -8.0000, A 0.000, B 0.000, C 0.000 }
gfCNCPoint5[29137] = {X 163.8528, Y 19.2746, Z -8.0000, A 0.000, B 0.000, C 0.000 }
gfCNCPoint5[29138] = {X 163.4280, Y 20.0990, Z -8.0000, A 0.000, B 0.000, C 0.000 }
gfCNCPoint5[29139] = {X 162.8549, Y 20.8281, Z -8.0000, A 0.000, B 0.000, C 0.000 }
gfCNCPoint5[29140] = {X 162.1542, Y 21.4357, Z -8.0000, A 0.000, B 0.000, C 0.000 }
gfCNCPoint5[29141] = {X 161.3512, Y 21.8997, Z -8.0000, A 0.000, B 0.000, C 0.000 }
gfCNCPoint5[29142] = {X 160.4749, Y 22.2034, Z -8.0000, A 0.000, B 0.000, C 0.000 }
gfCNCPoint5[29143] = {X 162.1759, Y 29.1996, Z -8.0000, A 0.000, B 0.000, C 0.000 }
gfCNCPoint5[29144] = {X 161.1136, Y 29.4080, Z -8.0000, A 0.000, B 0.000, C 0.000 }
gfCNCPoint5[29145] = {X 160.0370, Y 29.5204, Z -8.0000, A 0.000, B 0.000, C 0.000 }
gfCNCPoint5[29146] = {X 160.0366, Y 38.3362, Z -8.0000, A 0.000, B 0.000, C 0.000 }
gfCNCPoint5[29147] = {X 160.6847, Y 39.6934, Z -8.0000, A 0.000, B 0.000, C 0.000 }
gfCNCPoint5[29148] = {X 161.1595, Y 41.1206, Z -8.0000, A 0.000, B 0.000, C 0.000 }
gfCNCPoint5[29149] = {X 162.0518, Y 41.1205, Z -8.0000, A 0.000, B 0.000, C 0.000 }
gfCNCPoint5[29150] = {X 161.8695, Y 40.3467, Z -8.0000, A 0.000, B 0.000, C 0.000 }
gfCNCPoint5[29151] = {X 161.7169, Y 39.5666, Z -8.0000, A 0.000, B 0.000, C 0.000 }
gfCNCPoint5[29152] = {X 161.5938, Y 38.7932, Z -8.0000, A 0.000, B 0.000, C 0.000 }
gfCNCPoint5[29153] = {X 161.3791, Y 36.8687, Z -8.0000, A 0.000, B 0.000, C 0.000 }
gfCNCPoint5[29154] = {X 161.3302, Y 34.9328, Z -8.0000, A 0.000, B 0.000, C 0.000 }
gfCNCPoint5[29155] = {X 161.4475, Y 32.9999, Z -8.0000, A 0.000, B 0.000, C 0.000 }
gfCNCPoint5[29156] = {X 161.7301, Y 31.0841, Z -8.0000, A 0.000, B 0.000, C 0.000 }
gfCNCPoint5[29157] = {X 162.1759, Y 29.1996, Z -8.0000, A 0.000, B 0.000, C 0.000 }
gfCNCPoint5[29158] = {X 161.6089, Y 26.8675, Z -8.0000, A 0.000, B 0.000, C 0.000 }
gfCNCPoint5[29159] = {X 160.4737, Y 27.0728, Z -8.0000, A 0.000, B 0.000, C 0.000 }
gfCNCPoint5[29160] = {X 159.3221, Y 27.1415, Z -8.0000, A 0.000, B 0.000, C 0.000 }
gfCNCPoint5[29161] = {X 158.6622, Y 27.1415, Z -8.0000, A 0.000, B 0.000, C 0.000 }
gfCNCPoint5[29162] = {X 158.1489, Y 27.1263, Z -8.0000, A 0.000, B 0.000, C 0.000 }
gfCNCPoint5[29163] = {X 157.6371, Y 27.0839, Z -8.0000, A 0.000, B 0.000, C 0.000 }
gfCNCPoint5[29164] = {X 157.6365, Y 38.9958, Z -8.0000, A 0.000, B 0.000, C 0.000 }
gfCNCPoint5[29165] = {X 158.2204, Y 40.0482, Z -8.0000, A 0.000, B 0.000, C 0.000 }
gfCNCPoint5[29166] = {X 158.6695, Y 41.1647, Z -8.0000, A 0.000, B 0.000, C 0.000 }
gfCNCPoint5[29167] = {X 158.9769, Y 42.3282, Z -8.0000, A 0.000, B 0.000, C 0.000 }
gfCNCPoint5[29168] = {X 159.1379, Y 43.5209, Z -8.0000, A 0.000, B 0.000, C 0.000 }
gfCNCPoint5[29169] = {X 165.4258, Y 43.5200, Z -8.0000, A 0.000, B 0.000, C 0.000 }
gfCNCPoint5[29170] = {X 164.8366, Y 42.0454, Z -8.0000, A 0.000, B 0.000, C 0.000 }
gfCNCPoint5[29171] = {X 164.3769, Y 40.5255, Z -8.0000, A 0.000, B 0.000, C 0.000 }
gfCNCPoint5[29172] = {X 164.2176, Y 39.8500, Z -8.0000, A 0.000, B 0.000, C 0.000 }
gfCNCPoint5[29173] = {X 164.0838, Y 39.1689, Z -8.0000, A 0.000, B 0.000, C 0.000 }
gfCNCPoint5[29174] = {X 163.9647, Y 38.4207, Z -8.0000, A 0.000, B 0.000, C 0.000 }
gfCNCPoint5[29175] = {X 163.7485, Y 36.2699, Z -8.0000, A 0.000, B 0.000, C 0.000 }
gfCNCPoint5[29176] = {X 163.7638, Y 34.1082, Z -8.0000, A 0.000, B 0.000, C 0.000 }
gfCNCPoint5[29177] = {X 164.0104, Y 31.9607, Z -8.0000, A 0.000, B 0.000, C 0.000 }
gfCNCPoint5[29178] = {X 164.4855, Y 29.8518, Z -8.0000, A 0.000, B 0.000, C 0.000 }
gfCNCPoint5[29179] = {X 164.8364, Y 28.7346, Z -8.0000, A 0.000, B 0.000, C 0.000 }
gfCNCPoint5[29180] = {X 165.2515, Y 27.6396, Z -8.0000, A 0.000, B 0.000, C 0.000 }
gfCNCPoint5[29181] = {X 165.8682, Y 26.3072, Z -8.0000, A 0.000, B 0.000, C 0.000 }
gfCNCPoint5[29182] = {X 166.6029, Y 25.0360, Z -8.0000, A 0.000, B 0.000, C 0.000 }
gfCNCPoint5[29183] = {X 167.4497, Y 23.8365, Z -8.0000, A 0.000, B 0.000, C 0.000 }
gfCNCPoint5[29184] = {X 167.1640, Y 23.1367, Z -8.0000, A 0.000, B 0.000, C 0.000 }
gfCNCPoint5[29185] = {X 166.2875, Y 24.1836, Z -8.0000, A 0.000, B 0.000, C 0.000 }
gfCNCPoint5[29186] = {X 165.2724, Y 25.0968, Z -8.0000, A 0.000, B 0.000, C 0.000 }
gfCNCPoint5[29187] = {X 164.1389, Y 25.8580, Z -8.0000, A 0.000, B 0.000, C 0.000 }
gfCNCPoint5[29188] = {X 162.9096, Y 26.4522, Z -8.0000, A 0.000, B 0.000, C 0.000 }
gfCNCPoint5[29189] = {X 161.6089, Y 26.8675, Z -8.0000, A 0.000, B 0.000, C 0.000 }
gfCNCPoint5[29190] = {X 161.0419, Y 24.5355, Z -8.0000, A 0.000, B 0.000, C 0.000 }
gfCNCPoint5[29191] = {X 160.1882, Y 24.6898, Z -8.0000, A 0.000, B 0.000, C 0.000 }
gfCNCPoint5[29192] = {X 159.3221, Y 24.7415, Z -8.0000, A 0.000, B 0.000, C 0.000 }
gfCNCPoint5[29193] = {X 158.6699, Y 24.7415, Z -8.0000, A 0.000, B 0.000, C 0.000 }
gfCNCPoint5[29194] = {X 158.2835, Y 24.7301, Z -8.0000, A 0.000, B 0.000, C 0.000 }
gfCNCPoint5[29195] = {X 157.8982, Y 24.6982, Z -8.0000, A 0.000, B 0.000, C 0.000 }
gfCNCPoint5[29196] = {X 156.9783, Y 24.5375, Z -8.0000, A 0.000, B 0.000, C 0.000 }
gfCNCPoint5[29197] = {X 156.0865, Y 24.2609, Z -8.0000, A 0.000, B 0.000, C 0.000 }
gfCNCPoint5[29198] = {X 155.2372, Y 23.8728, Z -8.0000, A 0.000, B 0.000, C 0.000 }
gfCNCPoint5[29199] = {X 155.2365, Y 39.7518, Z -8.0000, A 0.000, B 0.000, C 0.000 }
gfCNCPoint5[29200] = {X 155.8272, Y 40.6433, Z -8.0000, A 0.000, B 0.000, C 0.000 }
gfCNCPoint5[29201] = {X 156.2813, Y 41.6115, Z -8.0000, A 0.000, B 0.000, C 0.000 }
gfCNCPoint5[29202] = {X 156.5892, Y 42.6357, Z -8.0000, A 0.000, B 0.000, C 0.000 }
gfCNCPoint5[29203] = {X 156.7441, Y 43.6938, Z -8.0000, A 0.000, B 0.000, C 0.000 }
gfCNCPoint5[29204] = {X 156.7580, Y 43.9467, Z -8.0000, A 0.000, B 0.000, C 0.000 }
gfCNCPoint5[29205] = {X 156.7631, Y 44.1999, Z -8.0000, A 0.000, B 0.000, C 0.000 }
gfCNCPoint5[29206] = {X 156.7628, Y 45.0700, Z -8.0000, A 0.000, B 0.000, C 0.000 }
gfCNCPoint5[29207] = {X 156.7347, Y 45.6426, Z -8.0000, A 0.000, B 0.000, C 0.000 }
gfCNCPoint5[29208] = {X 156.6616, Y 46.2112, Z -8.0000, A 0.000, B 0.000, C 0.000 }
gfCNCPoint5[29209] = {X 157.9054, Y 46.0005, Z -8.0000, A 0.000, B 0.000, C 0.000 }
gfCNCPoint5[29210] = {X 159.1644, Y 45.9207, Z -8.0000, A 0.000, B 0.000, C 0.000 }
gfCNCPoint5[29211] = {X 159.2312, Y 45.9202, Z -8.0000, A 0.000, B 0.000, C 0.000 }
gfCNCPoint5[29212] = {X 159.2980, Y 45.9200, Z -8.0000, A 0.000, B 0.000, C 0.000 }
gfCNCPoint5[29213] = {X 169.6787, Y 45.9200, Z -8.0000, A 0.000, B 0.000, C 0.000 }
gfCNCPoint5[29214] = {X 168.8976, Y 44.8498, Z -8.0000, A 0.000, B 0.000, C 0.000 }
gfCNCPoint5[29215] = {X 168.2078, Y 43.7186, Z -8.0000, A 0.000, B 0.000, C 0.000 }
gfCNCPoint5[29216] = {X 167.6139, Y 42.5342, Z -8.0000, A 0.000, B 0.000, C 0.000 }
gfCNCPoint5[29217] = {X 167.1231, Y 41.3128, Z -8.0000, A 0.000, B 0.000, C 0.000 }
gfCNCPoint5[29218] = {X 166.7344, Y 40.0552, Z -8.0000, A 0.000, B 0.000, C 0.000 }
gfCNCPoint5[29219] = {X 166.4505, Y 38.7698, Z -8.0000, A 0.000, B 0.000, C 0.000 }
gfCNCPoint5[29220] = {X 166.3357, Y 38.0485, Z -8.0000, A 0.000, B 0.000, C 0.000 }
gfCNCPoint5[29221] = {X 166.1443, Y 36.1221, Z -8.0000, A 0.000, B 0.000, C 0.000 }
gfCNCPoint5[29222] = {X 166.1636, Y 34.1864, Z -8.0000, A 0.000, B 0.000, C 0.000 }
gfCNCPoint5[29223] = {X 166.3935, Y 32.2642, Z -8.0000, A 0.000, B 0.000, C 0.000 }
gfCNCPoint5[29224] = {X 166.8312, Y 30.3785, Z -8.0000, A 0.000, B 0.000, C 0.000 }
gfCNCPoint5[29225] = {X 167.4715, Y 28.5516, Z -8.0000, A 0.000, B 0.000, C 0.000 }
gfCNCPoint5[29226] = {X 168.2321, Y 26.9815, Z -8.0000, A 0.000, B 0.000, C 0.000 }
gfCNCPoint5[29227] = {X 169.1845, Y 25.5199, Z -8.0000, A 0.000, B 0.000, C 0.000 }
gfCNCPoint5[29228] = {X 170.3136, Y 24.1899, Z -8.0000, A 0.000, B 0.000, C 0.000 }
gfCNCPoint5[29229] = {X 169.9862, Y 23.6218, Z -8.0000, A 0.000, B 0.000, C 0.000 }
gfCNCPoint5[29230] = {X 169.7113, Y 23.0265, Z -8.0000, A 0.000, B 0.000, C 0.000 }
gfCNCPoint5[29231] = {X 167.1001, Y 16.6309, Z -8.0000, A 0.000, B 0.000, C 0.000 }
gfCNCPoint5[29232] = {X 166.7820, Y 15.6636, Z -8.0000, A 0.000, B 0.000, C 0.000 }
gfCNCPoint5[29233] = {X 166.6021, Y 14.6613, Z -8.0000, A 0.000, B 0.000, C 0.000 }
gfCNCPoint5[29234] = {X 166.6021, Y 17.4615, Z -8.0000, A 0.000, B 0.000, C 0.000 }
gfCNCPoint5[29235] = {X 166.5130, Y 18.5970, Z -8.0000, A 0.000, B 0.000, C 0.000 }
gfCNCPoint5[29236] = {X 166.2479, Y 19.7047, Z -8.0000, A 0.000, B 0.000, C 0.000 }
gfCNCPoint5[29237] = {X 165.8132, Y 20.7575, Z -8.0000, A 0.000, B 0.000, C 0.000 }
gfCNCPoint5[29238] = {X 165.2197, Y 21.7296, Z -8.0000, A 0.000, B 0.000, C 0.000 }
gfCNCPoint5[29239] = {X 164.3789, Y 22.6987, Z -8.0000, A 0.000, B 0.000, C 0.000 }
gfCNCPoint5[29240] = {X 163.3810, Y 23.5050, Z -8.0000, A 0.000, B 0.000, C 0.000 }
gfCNCPoint5[29241] = {X 162.2570, Y 24.1237, Z -8.0000, A 0.000, B 0.000, C 0.000 }
gfCNCPoint5[29242] = {X 161.0419, Y 24.5355, Z -8.0000, A 0.000, B 0.000, C 0.000 }
gfCNCPoint5[29243] = {X 160.4749, Y 22.2034, Z -8.0000, A 0.000, B 0.000, C 0.000 }
gfCNCPoint5[29244] = {X 159.9026, Y 22.3069, Z -8.0000, A 0.000, B 0.000, C 0.000 }
gfCNCPoint5[29245] = {X 159.3221, Y 22.3415, Z -8.0000, A 0.000, B 0.000, C 0.000 }
gfCNCPoint5[29246] = {X 158.6776, Y 22.3415, Z -8.0000, A 0.000, B 0.000, C 0.000 }
gfCNCPoint5[29247] = {X 157.8807, Y 22.2738, Z -8.0000, A 0.000, B 0.000, C 0.000 }
gfCNCPoint5[29248] = {X 157.1053, Y 22.0776, Z -8.0000, A 0.000, B 0.000, C 0.000 }
gfCNCPoint5[29249] = {X 156.3721, Y 21.7581, Z -8.0000, A 0.000, B 0.000, C 0.000 }
gfCNCPoint5[29250] = {X 155.5228, Y 21.1803, Z -8.0000, A 0.000, B 0.000, C 0.000 }
gfCNCPoint5[29251] = {X 154.8123, Y 20.4383, Z -8.0000, A 0.000, B 0.000, C 0.000 }
gfCNCPoint5[29252] = {X 152.8374, Y 20.4389, Z -8.0000, A 0.000, B 0.000, C 0.000 }
gfCNCPoint5[29253] = {X 152.8364, Y 40.6543, Z -8.0000, A 0.000, B 0.000, C 0.000 }
gfCNCPoint5[29254] = {X 153.1745, Y 41.0198, Z -8.0000, A 0.000, B 0.000, C 0.000 }
gfCNCPoint5[29255] = {X 153.6802, Y 41.7242, Z -8.0000, A 0.000, B 0.000, C 0.000 }
gfCNCPoint5[29256] = {X 154.0540, Y 42.5068, Z -8.0000, A 0.000, B 0.000, C 0.000 }
gfCNCPoint5[29257] = {X 154.2840, Y 43.3429, Z -8.0000, A 0.000, B 0.000, C 0.000 }
gfCNCPoint5[29258] = {X 154.3631, Y 44.2065, Z -8.0000, A 0.000, B 0.000, C 0.000 }
gfCNCPoint5[29259] = {X 154.3629, Y 45.0469, Z -8.0000, A 0.000, B 0.000, C 0.000 }
gfCNCPoint5[29260] = {X 154.3440, Y 45.4308, Z -8.0000, A 0.000, B 0.000, C 0.000 }
gfCNCPoint5[29261] = {X 154.2951, Y 45.8119, Z -8.0000, A 0.000, B 0.000, C 0.000 }
gfCNCPoint5[29262] = {X 154.0370, Y 46.7541, Z -8.0000, A 0.000, B 0.000, C 0.000 }
gfCNCPoint5[29263] = {X 153.5963, Y 47.6260, Z -8.0000, A 0.000, B 0.000, C 0.000 }
gfCNCPoint5[29264] = {X 152.9909, Y 48.3926, Z -8.0000, A 0.000, B 0.000, C 0.000 }
gfCNCPoint5[29265] = {X 152.2448, Y 49.0233, Z -8.0000, A 0.000, B 0.000, C 0.000 }
gfCNCPoint5[29266] = {X 151.3881, Y 49.4928, Z -8.0000, A 0.000, B 0.000, C 0.000 }
gfCNCPoint5[29267] = {X 150.4551, Y 49.7822, Z -8.0000, A 0.000, B 0.000, C 0.000 }
gfCNCPoint5[29268] = {X 149.4831, Y 49.8800, Z -8.0000, A 0.000, B 0.000, C 0.000 }
gfCNCPoint5[29269] = {X 143.0396, Y 49.8800, Z -8.0000, A 0.000, B 0.000, C 0.000 }
gfCNCPoint5[29270] = {X 142.0923, Y 49.7872, Z -8.0000, A 0.000, B 0.000, C 0.000 }
gfCNCPoint5[29271] = {X 141.1811, Y 49.5122, Z -8.0000, A 0.000, B 0.000, C 0.000 }
gfCNCPoint5[29272] = {X 140.3405, Y 49.0656, Z -8.0000, A 0.000, B 0.000, C 0.000 }
gfCNCPoint5[29273] = {X 139.6026, Y 48.4643, Z -8.0000, A 0.000, B 0.000, C 0.000 }
gfCNCPoint5[29274] = {X 138.9955, Y 47.7312, Z -8.0000, A 0.000, B 0.000, C 0.000 }
gfCNCPoint5[29275] = {X 138.5423, Y 46.8942, Z -8.0000, A 0.000, B 0.000, C 0.000 }
gfCNCPoint5[29276] = {X 138.2601, Y 45.9852, Z -8.0000, A 0.000, B 0.000, C 0.000 }
gfCNCPoint5[29277] = {X 138.1598, Y 45.0386, Z -8.0000, A 0.000, B 0.000, C 0.000 }
gfCNCPoint5[29278] = {X 138.1601, Y 44.1417, Z -8.0000, A 0.000, B 0.000, C 0.000 }
gfCNCPoint5[29279] = {X 138.2148, Y 43.4769, Z -8.0000, A 0.000, B 0.000, C 0.000 }
gfCNCPoint5[29280] = {X 138.3597, Y 42.8258, Z -8.0000, A 0.000, B 0.000, C 0.000 }
gfCNCPoint5[29281] = {X 129.1532, Y 40.1052, Z -8.0000, A 0.000, B 0.000, C 0.000 }
gfCNCPoint5[29282] = {X 129.5665, Y 38.9035, Z -8.0000, A 0.000, B 0.000, C 0.000 }
gfCNCPoint5[29283] = {X 130.0836, Y 37.7426, Z -8.0000, A 0.000, B 0.000, C 0.000 }
gfCNCPoint5[29284] = {X 130.0836, Y 31.6021, Z -8.0000, A 0.000, B 0.000, C 0.000 }
gfCNCPoint5[29285] = {X 129.2066, Y 31.3798, Z -8.0000, A 0.000, B 0.000, C 0.000 }
gfCNCPoint5[29286] = {X 128.3452, Y 31.1032, Z -8.0000, A 0.000, B 0.000, C 0.000 }
gfCNCPoint5[29287] = {X 128.3453, Y 38.3312, Z -8.0000, A 0.000, B 0.000, C 0.000 }
gfCNCPoint5[29288] = {X 128.7851, Y 39.2019, Z -8.0000, A 0.000, B 0.000, C 0.000 }
gfCNCPoint5[29289] = {X 129.1532, Y 40.1052, Z -8.0000, A 0.000, B 0.000, C 0.000 }
gfCNCPoint5[29290] = {X 131.4548, Y 40.7854, Z -8.0000, A 0.000, B 0.000, C 0.000 }
gfCNCPoint5[29291] = {X 131.9017, Y 39.5320, Z -8.0000, A 0.000, B 0.000, C 0.000 }
gfCNCPoint5[29292] = {X 132.4836, Y 38.3354, Z -8.0000, A 0.000, B 0.000, C 0.000 }
gfCNCPoint5[29293] = {X 132.4836, Y 29.5202, Z -8.0000, A 0.000, B 0.000, C 0.000 }
gfCNCPoint5[29294] = {X 131.3527, Y 29.3994, Z -8.0000, A 0.000, B 0.000, C 0.000 }
gfCNCPoint5[29295] = {X 130.2382, Y 29.1727, Z -8.0000, A 0.000, B 0.000, C 0.000 }
gfCNCPoint5[29296] = {X 129.1500, Y 28.8422, Z -8.0000, A 0.000, B 0.000, C 0.000 }
gfCNCPoint5[29297] = {X 128.0256, Y 28.3769, Z -8.0000, A 0.000, B 0.000, C 0.000 }
gfCNCPoint5[29298] = {X 126.9537, Y 27.8009, Z -8.0000, A 0.000, B 0.000, C 0.000 }
gfCNCPoint5[29299] = {X 125.9452, Y 27.1200, Z -8.0000, A 0.000, B 0.000, C 0.000 }
gfCNCPoint5[29300] = {X 125.9453, Y 38.9915, Z -8.0000, A 0.000, B 0.000, C 0.000 }
gfCNCPoint5[29301] = {X 126.4743, Y 39.9295, Z -8.0000, A 0.000, B 0.000, C 0.000 }
gfCNCPoint5[29302] = {X 126.8960, Y 40.9205, Z -8.0000, A 0.000, B 0.000, C 0.000 }
gfCNCPoint5[29303] = {X 127.2098, Y 41.9730, Z -8.0000, A 0.000, B 0.000, C 0.000 }
gfCNCPoint5[29304] = {X 127.4025, Y 43.0542, Z -8.0000, A 0.000, B 0.000, C 0.000 }
gfCNCPoint5[29305] = {X 127.4714, Y 44.1502, Z -8.0000, A 0.000, B 0.000, C 0.000 }
gfCNCPoint5[29306] = {X 127.4716, Y 45.0000, Z -8.0000, A 0.000, B 0.000, C 0.000 }
gfCNCPoint5[29307] = {X 127.4070, Y 46.1159, Z -8.0000, A 0.000, B 0.000, C 0.000 }
gfCNCPoint5[29308] = {X 127.2143, Y 47.2168, Z -8.0000, A 0.000, B 0.000, C 0.000 }
gfCNCPoint5[29309] = {X 126.8960, Y 48.2883, Z -8.0000, A 0.000, B 0.000, C 0.000 }
gfCNCPoint5[29310] = {X 126.2883, Y 49.6376, Z -8.0000, A 0.000, B 0.000, C 0.000 }
gfCNCPoint5[29311] = {X 125.4821, Y 50.8786, Z -8.0000, A 0.000, B 0.000, C 0.000 }
gfCNCPoint5[29312] = {X 124.4962, Y 51.9821, Z -8.0000, A 0.000, B 0.000, C 0.000 }
gfCNCPoint5[29313] = {X 123.3536, Y 52.9225, Z -8.0000, A 0.000, B 0.000, C 0.000 }
gfCNCPoint5[29314] = {X 122.0810, Y 53.6778, Z -8.0000, A 0.000, B 0.000, C 0.000 }
gfCNCPoint5[29315] = {X 120.7081, Y 54.2302, Z -8.0000, A 0.000, B 0.000, C 0.000 }
gfCNCPoint5[29316] = {X 119.2671, Y 54.5669, Z -8.0000, A 0.000, B 0.000, C 0.000 }
gfCNCPoint5[29317] = {X 117.7916, Y 54.6800, Z -8.0000, A 0.000, B 0.000, C 0.000 }
gfCNCPoint5[29318] = {X 111.9185, Y 54.6800, Z -8.0000, A 0.000, B 0.000, C 0.000 }
gfCNCPoint5[29319] = {X 111.7456, Y 54.6785, Z -8.0000, A 0.000, B 0.000, C 0.000 }
gfCNCPoint5[29320] = {X 111.5728, Y 54.6738, Z -8.0000, A 0.000, B 0.000, C 0.000 }
gfCNCPoint5[29321] = {X 111.0585, Y 69.0646, Z -8.0000, A 0.000, B 0.000, C 0.000 }
gfCNCPoint5[29322] = {X 109.0296, Y 68.9061, Z -8.0000, A 0.000, B 0.000, C 0.000 }
gfCNCPoint5[29323] = {X 107.0213, Y 68.5768, Z -8.0000, A 0.000, B 0.000, C 0.000 }
gfCNCPoint5[29324] = {X 105.0765, Y 68.8983, Z -8.0000, A 0.000, B 0.000, C 0.000 }
gfCNCPoint5[29325] = {X 103.1119, Y 69.0597, Z -8.0000, A 0.000, B 0.000, C 0.000 }
gfCNCPoint5[29326] = {X 101.1407, Y 69.0599, Z -8.0000, A 0.000, B 0.000, C 0.000 }
gfCNCPoint5[29327] = {X 99.1761, Y 68.8989, Z -8.0000, A 0.000, B 0.000, C 0.000 }
gfCNCPoint5[29328] = {X 97.2313, Y 68.5777, Z -8.0000, A 0.000, B 0.000, C 0.000 }
gfCNCPoint5[29329] = {X 95.6131, Y 68.8563, Z -8.0000, A 0.000, B 0.000, C 0.000 }
gfCNCPoint5[29330] = {X 93.9796, Y 69.0240, Z -8.0000, A 0.000, B 0.000, C 0.000 }
gfCNCPoint5[29331] = {X 92.3385, Y 69.0800, Z -8.0000, A 0.000, B 0.000, C 0.000 }
gfCNCPoint5[29332] = {X 86.6884, Y 69.0800, Z -8.0000, A 0.000, B 0.000, C 0.000 }
gfCNCPoint5[29333] = {X 84.7315, Y 70.2669, Z -8.0000, A 0.000, B 0.000, C 0.000 }
gfCNCPoint5[29334] = {X 82.6867, Y 71.2952, Z -8.0000, A 0.000, B 0.000, C 0.000 }
gfCNCPoint5[29335] = {X 107.2713, Y 71.2952, Z -8.0000, A 0.000, B 0.000, C 0.000 }
gfCNCPoint5[29336] = {X 109.1257, Y 70.1133, Z -8.0000, A 0.000, B 0.000, C 0.000 }
gfCNCPoint5[29337] = {X 111.0585, Y 69.0646, Z -8.0000, A 0.000, B 0.000, C 0.000 }
gfCNCPoint5[29338] = {X 111.1442, Y 66.6662, Z -8.0000, A 0.000, B 0.000, C 0.000 }
gfCNCPoint5[29339] = {X 109.0696, Y 66.4920, Z -8.0000, A 0.000, B 0.000, C 0.000 }
gfCNCPoint5[29340] = {X 107.0213, Y 66.1197, Z -8.0000, A 0.000, B 0.000, C 0.000 }
gfCNCPoint5[29341] = {X 105.0796, Y 66.4776, Z -8.0000, A 0.000, B 0.000, C 0.000 }
gfCNCPoint5[29342] = {X 103.1135, Y 66.6574, Z -8.0000, A 0.000, B 0.000, C 0.000 }
gfCNCPoint5[29343] = {X 101.1392, Y 66.6576, Z -8.0000, A 0.000, B 0.000, C 0.000 }
gfCNCPoint5[29344] = {X 99.1730, Y 66.4782, Z -8.0000, A 0.000, B 0.000, C 0.000 }
gfCNCPoint5[29345] = {X 97.2313, Y 66.1207, Z -8.0000, A 0.000, B 0.000, C 0.000 }
gfCNCPoint5[29346] = {X 95.6161, Y 66.4308, Z -8.0000, A 0.000, B 0.000, C 0.000 }
gfCNCPoint5[29347] = {X 93.9821, Y 66.6176, Z -8.0000, A 0.000, B 0.000, C 0.000 }
gfCNCPoint5[29348] = {X 92.3385, Y 66.6800, Z -8.0000, A 0.000, B 0.000, C 0.000 }
gfCNCPoint5[29349] = {X 85.9487, Y 66.6800, Z -8.0000, A 0.000, B 0.000, C 0.000 }
gfCNCPoint5[29350] = {X 83.8778, Y 67.9936, Z -8.0000, A 0.000, B 0.000, C 0.000 }
gfCNCPoint5[29351] = {X 81.6943, Y 69.1100, Z -8.0000, A 0.000, B 0.000, C 0.000 }
gfCNCPoint5[29352] = {X 79.6014, Y 69.9549, Z -8.0000, A 0.000, B 0.000, C 0.000 }
gfCNCPoint5[29353] = {X 77.4441, Y 70.6185, Z -8.0000, A 0.000, B 0.000, C 0.000 }
gfCNCPoint5[29354] = {X 75.2381, Y 71.0959, Z -8.0000, A 0.000, B 0.000, C 0.000 }
gfCNCPoint5[29355] = {X 72.9995, Y 71.3838, Z -8.0000, A 0.000, B 0.000, C 0.000 }
gfCNCPoint5[29356] = {X 70.7445, Y 71.4800, Z -8.0000, A 0.000, B 0.000, C 0.000 }
gfCNCPoint5[29357] = {X 64.1851, Y 71.4800, Z -8.0000, A 0.000, B 0.000, C 0.000 }
gfCNCPoint5[29358] = {X 62.0752, Y 71.3958, Z -8.0000, A 0.000, B 0.000, C 0.000 }
gfCNCPoint5[29359] = {X 59.9787, Y 71.1438, Z -8.0000, A 0.000, B 0.000, C 0.000 }
gfCNCPoint5[29360] = {X 57.9089, Y 70.7255, Z -8.0000, A 0.000, B 0.000, C 0.000 }
gfCNCPoint5[29361] = {X 55.8790, Y 70.1436, Z -8.0000, A 0.000, B 0.000, C 0.000 }
gfCNCPoint5[29362] = {X 53.8492, Y 70.7255, Z -8.0000, A 0.000, B 0.000, C 0.000 }
gfCNCPoint5[29363] = {X 51.7794, Y 71.1438, Z -8.0000, A 0.000, B 0.000, C 0.000 }
gfCNCPoint5[29364] = {X 49.6829, Y 71.3958, Z -8.0000, A 0.000, B 0.000, C 0.000 }
gfCNCPoint5[29365] = {X 47.5729, Y 71.4800, Z -8.0000, A 0.000, B 0.000, C 0.000 }
gfCNCPoint5[29366] = {X 40.6393, Y 71.4800, Z -8.0000, A 0.000, B 0.000, C 0.000 }
gfCNCPoint5[29367] = {X 38.8062, Y 71.4165, Z -8.0000, A 0.000, B 0.000, C 0.000 }
gfCNCPoint5[29368] = {X 36.9818, Y 71.2262, Z -8.0000, A 0.000, B 0.000, C 0.000 }
gfCNCPoint5[29369] = {X 34.3986, Y 72.0364, Z -8.0000, A 0.000, B 0.000, C 0.000 }
gfCNCPoint5[29370] = {X 31.7542, Y 72.6168, Z -8.0000, A 0.000, B 0.000, C 0.000 }
gfCNCPoint5[29371] = {X 30.3314, Y 73.1755, Z -8.0000, A 0.000, B 0.000, C 0.000 }
gfCNCPoint5[29372] = {X 28.8938, Y 73.6952, Z -8.0000, A 0.000, B 0.000, C 0.000 }
gfCNCPoint5[29373] = {X 108.0335, Y 73.6952, Z -8.0000, A 0.000, B 0.000, C 0.000 }
gfCNCPoint5[29374] = {X 110.0293, Y 72.3691, Z -8.0000, A 0.000, B 0.000, C 0.000 }
gfCNCPoint5[29375] = {X 112.1282, Y 71.2131, Z -8.0000, A 0.000, B 0.000, C 0.000 }
gfCNCPoint5[29376] = {X 113.1244, Y 70.7406, Z -8.0000, A 0.000, B 0.000, C 0.000 }
gfCNCPoint5[29377] = {X 114.1380, Y 70.3064, Z -8.0000, A 0.000, B 0.000, C 0.000 }
gfCNCPoint5[29378] = {X 117.4405, Y 66.6800, Z -8.0000, A 0.000, B 0.000, C 0.000 }
gfCNCPoint5[29379] = {X 111.9185, Y 66.6800, Z -8.0000, A 0.000, B 0.000, C 0.000 }
gfCNCPoint5[29380] = {X 111.5313, Y 66.6765, Z -8.0000, A 0.000, B 0.000, C 0.000 }
gfCNCPoint5[29381] = {X 111.1442, Y 66.6662, Z -8.0000, A 0.000, B 0.000, C 0.000 }
gfCNCPoint5[29382] = {X 111.2299, Y 64.2677, Z -8.0000, A 0.000, B 0.000, C 0.000 }
gfCNCPoint5[29383] = {X 109.1084, Y 64.0741, Z -8.0000, A 0.000, B 0.000, C 0.000 }
gfCNCPoint5[29384] = {X 107.0213, Y 63.6477, Z -8.0000, A 0.000, B 0.000, C 0.000 }
gfCNCPoint5[29385] = {X 105.0841, Y 64.0514, Z -8.0000, A 0.000, B 0.000, C 0.000 }
gfCNCPoint5[29386] = {X 103.1158, Y 64.2545, Z -8.0000, A 0.000, B 0.000, C 0.000 }
gfCNCPoint5[29387] = {X 101.1370, Y 64.2547, Z -8.0000, A 0.000, B 0.000, C 0.000 }
gfCNCPoint5[29388] = {X 99.1686, Y 64.0521, Z -8.0000, A 0.000, B 0.000, C 0.000 }
gfCNCPoint5[29389] = {X 97.2313, Y 63.6488, Z -8.0000, A 0.000, B 0.000, C 0.000 }
gfCNCPoint5[29390] = {X 95.6204, Y 63.9986, Z -8.0000, A 0.000, B 0.000, C 0.000 }
gfCNCPoint5[29391] = {X 93.9855, Y 64.2095, Z -8.0000, A 0.000, B 0.000, C 0.000 }
gfCNCPoint5[29392] = {X 92.3385, Y 64.2800, Z -8.0000, A 0.000, B 0.000, C 0.000 }
gfCNCPoint5[29393] = {X 85.8951, Y 64.2800, Z -8.0000, A 0.000, B 0.000, C 0.000 }
gfCNCPoint5[29394] = {X 85.5417, Y 64.2768, Z -8.0000, A 0.000, B 0.000, C 0.000 }
gfCNCPoint5[29395] = {X 85.1884, Y 64.2670, Z -8.0000, A 0.000, B 0.000, C 0.000 }
gfCNCPoint5[29396] = {X 83.3593, Y 65.5113, Z -8.0000, A 0.000, B 0.000, C 0.000 }
gfCNCPoint5[29397] = {X 81.4238, Y 66.5824, Z -8.0000, A 0.000, B 0.000, C 0.000 }
gfCNCPoint5[29398] = {X 79.3981, Y 67.4713, Z -8.0000, A 0.000, B 0.000, C 0.000 }
gfCNCPoint5[29399] = {X 77.2994, Y 68.1706, Z -8.0000, A 0.000, B 0.000, C 0.000 }
gfCNCPoint5[29400] = {X 75.1454, Y 68.6744, Z -8.0000, A 0.000, B 0.000, C 0.000 }
gfCNCPoint5[29401] = {X 72.9543, Y 68.9784, Z -8.0000, A 0.000, B 0.000, C 0.000 }
gfCNCPoint5[29402] = {X 70.7445, Y 69.0800, Z -8.0000, A 0.000, B 0.000, C 0.000 }
gfCNCPoint5[29403] = {X 64.1851, Y 69.0800, Z -8.0000, A 0.000, B 0.000, C 0.000 }
gfCNCPoint5[29404] = {X 62.0678, Y 68.9867, Z -8.0000, A 0.000, B 0.000, C 0.000 }
gfCNCPoint5[29405] = {X 59.9669, Y 68.7076, Z -8.0000, A 0.000, B 0.000, C 0.000 }
gfCNCPoint5[29406] = {X 57.8986, Y 68.2449, Z -8.0000, A 0.000, B 0.000, C 0.000 }
gfCNCPoint5[29407] = {X 55.8790, Y 67.6021, Z -8.0000, A 0.000, B 0.000, C 0.000 }
gfCNCPoint5[29408] = {X 53.8595, Y 68.2449, Z -8.0000, A 0.000, B 0.000, C 0.000 }
gfCNCPoint5[29409] = {X 51.7912, Y 68.7076, Z -8.0000, A 0.000, B 0.000, C 0.000 }
gfCNCPoint5[29410] = {X 49.6903, Y 68.9867, Z -8.0000, A 0.000, B 0.000, C 0.000 }
gfCNCPoint5[29411] = {X 47.5729, Y 69.0800, Z -8.0000, A 0.000, B 0.000, C 0.000 }
gfCNCPoint5[29412] = {X 40.6393, Y 69.0800, Z -8.0000, A 0.000, B 0.000, C 0.000 }
gfCNCPoint5[29413] = {X 38.6756, Y 68.9998, Z -8.0000, A 0.000, B 0.000, C 0.000 }
gfCNCPoint5[29414] = {X 36.7249, Y 68.7597, Z -8.0000, A 0.000, B 0.000, C 0.000 }
gfCNCPoint5[29415] = {X 34.8830, Y 69.4002, Z -8.0000, A 0.000, B 0.000, C 0.000 }
gfCNCPoint5[29416] = {X 33.0015, Y 69.9128, Z -8.0000, A 0.000, B 0.000, C 0.000 }
gfCNCPoint5[29417] = {X 31.0892, Y 70.2952, Z -8.0000, A 0.000, B 0.000, C 0.000 }
gfCNCPoint5[29418] = {X 29.6075, Y 70.8834, Z -8.0000, A 0.000, B 0.000, C 0.000 }
gfCNCPoint5[29419] = {X 28.1088, Y 71.4272, Z -8.0000, A 0.000, B 0.000, C 0.000 }
gfCNCPoint5[29420] = {X 27.6142, Y 71.5956, Z -8.0000, A 0.000, B 0.000, C 0.000 }
gfCNCPoint5[29421] = {X 27.1180, Y 71.7593, Z -8.0000, A 0.000, B 0.000, C 0.000 }
gfCNCPoint5[29422] = {X 25.5190, Y 72.2532, Z -8.0000, A 0.000, B 0.000, C 0.000 }
gfCNCPoint5[29423] = {X 23.9033, Y 72.6897, Z -8.0000, A 0.000, B 0.000, C 0.000 }
gfCNCPoint5[29424] = {X 23.9033, Y 76.0952, Z -8.0000, A 0.000, B 0.000, C 0.000 }
gfCNCPoint5[29425] = {X 108.8316, Y 76.0952, Z -8.0000, A 0.000, B 0.000, C 0.000 }
gfCNCPoint5[29426] = {X 110.4007, Y 74.9741, Z -8.0000, A 0.000, B 0.000, C 0.000 }
gfCNCPoint5[29427] = {X 112.0471, Y 73.9702, Z -8.0000, A 0.000, B 0.000, C 0.000 }
gfCNCPoint5[29428] = {X 113.7623, Y 73.0888, Z -8.0000, A 0.000, B 0.000, C 0.000 }
gfCNCPoint5[29429] = {X 115.5371, Y 72.3345, Z -8.0000, A 0.000, B 0.000, C 0.000 }
gfCNCPoint5[29430] = {X 123.7242, Y 63.3445, Z -8.0000, A 0.000, B 0.000, C 0.000 }
gfCNCPoint5[29431] = {X 121.7828, Y 63.8624, Z -8.0000, A 0.000, B 0.000, C 0.000 }
gfCNCPoint5[29432] = {X 119.7981, Y 64.1753, Z -8.0000, A 0.000, B 0.000, C 0.000 }
gfCNCPoint5[29433] = {X 117.7916, Y 64.2800, Z -8.0000, A 0.000, B 0.000, C 0.000 }
gfCNCPoint5[29434] = {X 111.9185, Y 64.2800, Z -8.0000, A 0.000, B 0.000, C 0.000 }
gfCNCPoint5[29435] = {X 111.5741, Y 64.2769, Z -8.0000, A 0.000, B 0.000, C 0.000 }
gfCNCPoint5[29436] = {X 111.2299, Y 64.2677, Z -8.0000, A 0.000, B 0.000, C 0.000 }
gfCNCPoint5[29437] = {X 111.3156, Y 61.8692, Z -8.0000, A 0.000, B 0.000, C 0.000 }
gfCNCPoint5[29438] = {X 109.8654, Y 61.7547, Z -8.0000, A 0.000, B 0.000, C 0.000 }
gfCNCPoint5[29439] = {X 108.4304, Y 61.5157, Z -8.0000, A 0.000, B 0.000, C 0.000 }
gfCNCPoint5[29440] = {X 107.0213, Y 61.1540, Z -8.0000, A 0.000, B 0.000, C 0.000 }
gfCNCPoint5[29441] = {X 105.0907, Y 61.6173, Z -8.0000, A 0.000, B 0.000, C 0.000 }
gfCNCPoint5[29442] = {X 103.1191, Y 61.8506, Z -8.0000, A 0.000, B 0.000, C 0.000 }
gfCNCPoint5[29443] = {X 101.1337, Y 61.8509, Z -8.0000, A 0.000, B 0.000, C 0.000 }
gfCNCPoint5[29444] = {X 99.1620, Y 61.6181, Z -8.0000, A 0.000, B 0.000, C 0.000 }
gfCNCPoint5[29445] = {X 97.2313, Y 61.1553, Z -8.0000, A 0.000, B 0.000, C 0.000 }
gfCNCPoint5[29446] = {X 95.6267, Y 61.5566, Z -8.0000, A 0.000, B 0.000, C 0.000 }
gfCNCPoint5[29447] = {X 93.9906, Y 61.7990, Z -8.0000, A 0.000, B 0.000, C 0.000 }
gfCNCPoint5[29448] = {X 92.3385, Y 61.8800, Z -8.0000, A 0.000, B 0.000, C 0.000 }
gfCNCPoint5[29449] = {X 85.8951, Y 61.8800, Z -8.0000, A 0.000, B 0.000, C 0.000 }
gfCNCPoint5[29450] = {X 85.1609, Y 61.8640, Z -8.0000, A 0.000, B 0.000, C 0.000 }
gfCNCPoint5[29451] = {X 84.4280, Y 61.8161, Z -8.0000, A 0.000, B 0.000, C 0.000 }
gfCNCPoint5[29452] = {X 82.7247, Y 63.0692, Z -8.0000, A 0.000, B 0.000, C 0.000 }
gfCNCPoint5[29453] = {X 80.9073, Y 64.1504, Z -8.0000, A 0.000, B 0.000, C 0.000 }
gfCNCPoint5[29454] = {X 78.9932, Y 65.0494, Z -8.0000, A 0.000, B 0.000, C 0.000 }
gfCNCPoint5[29455] = {X 77.0007, Y 65.7577, Z -8.0000, A 0.000, B 0.000, C 0.000 }
gfCNCPoint5[29456] = {X 74.9487, Y 66.2685, Z -8.0000, A 0.000, B 0.000, C 0.000 }
gfCNCPoint5[29457] = {X 72.8566, Y 66.5769, Z -8.0000, A 0.000, B 0.000, C 0.000 }
gfCNCPoint5[29458] = {X 70.7445, Y 66.6800, Z -8.0000, A 0.000, B 0.000, C 0.000 }
gfCNCPoint5[29459] = {X 64.1851, Y 66.6800, Z -8.0000, A 0.000, B 0.000, C 0.000 }
gfCNCPoint5[29460] = {X 62.0576, Y 66.5754, Z -8.0000, A 0.000, B 0.000, C 0.000 }
gfCNCPoint5[29461] = {X 59.9505, Y 66.2624, Z -8.0000, A 0.000, B 0.000, C 0.000 }
gfCNCPoint5[29462] = {X 57.8844, Y 65.7442, Z -8.0000, A 0.000, B 0.000, C 0.000 }
gfCNCPoint5[29463] = {X 55.8790, Y 65.0258, Z -8.0000, A 0.000, B 0.000, C 0.000 }
gfCNCPoint5[29464] = {X 53.8737, Y 65.7442, Z -8.0000, A 0.000, B 0.000, C 0.000 }
gfCNCPoint5[29465] = {X 51.8075, Y 66.2624, Z -8.0000, A 0.000, B 0.000, C 0.000 }
gfCNCPoint5[29466] = {X 49.7005, Y 66.5754, Z -8.0000, A 0.000, B 0.000, C 0.000 }
gfCNCPoint5[29467] = {X 47.5729, Y 66.6800, Z -8.0000, A 0.000, B 0.000, C 0.000 }
gfCNCPoint5[29468] = {X 40.6393, Y 66.6800, Z -8.0000, A 0.000, B 0.000, C 0.000 }
gfCNCPoint5[29469] = {X 38.5455, Y 66.5787, Z -8.0000, A 0.000, B 0.000, C 0.000 }
gfCNCPoint5[29470] = {X 36.4714, Y 66.2756, Z -8.0000, A 0.000, B 0.000, C 0.000 }
gfCNCPoint5[29471] = {X 34.5050, Y 67.0024, Z -8.0000, A 0.000, B 0.000, C 0.000 }
gfCNCPoint5[29472] = {X 32.4865, Y 67.5684, Z -8.0000, A 0.000, B 0.000, C 0.000 }
gfCNCPoint5[29473] = {X 30.4290, Y 67.9701, Z -8.0000, A 0.000, B 0.000, C 0.000 }
gfCNCPoint5[29474] = {X 28.4170, Y 68.7669, Z -8.0000, A 0.000, B 0.000, C 0.000 }
gfCNCPoint5[29475] = {X 26.3732, Y 69.4778, Z -8.0000, A 0.000, B 0.000, C 0.000 }
gfCNCPoint5[29476] = {X 23.9567, Y 70.1968, Z -8.0000, A 0.000, B 0.000, C 0.000 }
gfCNCPoint5[29477] = {X 21.5033, Y 70.7776, Z -8.0000, A 0.000, B 0.000, C 0.000 }
gfCNCPoint5[29478] = {X 21.5033, Y 78.4952, Z -8.0000, A 0.000, B 0.000, C 0.000 }
gfCNCPoint5[29479] = {X 109.6712, Y 78.4952, Z -8.0000, A 0.000, B 0.000, C 0.000 }
gfCNCPoint5[29480] = {X 111.3416, Y 77.2343, Z -8.0000, A 0.000, B 0.000, C 0.000 }
gfCNCPoint5[29481] = {X 113.1153, Y 76.1232, Z -8.0000, A 0.000, B 0.000, C 0.000 }
gfCNCPoint5[29482] = {X 114.9787, Y 75.1703, Z -8.0000, A 0.000, B 0.000, C 0.000 }
gfCNCPoint5[29483] = {X 116.9178, Y 74.3828, Z -8.0000, A 0.000, B 0.000, C 0.000 }
gfCNCPoint5[29484] = {X 130.4100, Y 59.5675, Z -8.0000, A 0.000, B 0.000, C 0.000 }
gfCNCPoint5[29485] = {X 129.5273, Y 58.7526, Z -8.0000, A 0.000, B 0.000, C 0.000 }
gfCNCPoint5[29486] = {X 128.6970, Y 57.8844, Z -8.0000, A 0.000, B 0.000, C 0.000 }
gfCNCPoint5[29487] = {X 127.3923, Y 58.8838, Z -8.0000, A 0.000, B 0.000, C 0.000 }
gfCNCPoint5[29488] = {X 125.9965, Y 59.7517, Z -8.0000, A 0.000, B 0.000, C 0.000 }
gfCNCPoint5[29489] = {X 124.5230, Y 60.4797, Z -8.0000, A 0.000, B 0.000, C 0.000 }
gfCNCPoint5[29490] = {X 122.9857, Y 61.0610, Z -8.0000, A 0.000, B 0.000, C 0.000 }
gfCNCPoint5[29491] = {X 121.2860, Y 61.5143, Z -8.0000, A 0.000, B 0.000, C 0.000 }
gfCNCPoint5[29492] = {X 119.5483, Y 61.7883, Z -8.0000, A 0.000, B 0.000, C 0.000 }
gfCNCPoint5[29493] = {X 117.7916, Y 61.8800, Z -8.0000, A 0.000, B 0.000, C 0.000 }
gfCNCPoint5[29494] = {X 111.9185, Y 61.8800, Z -8.0000, A 0.000, B 0.000, C 0.000 }
gfCNCPoint5[29495] = {X 111.6170, Y 61.8773, Z -8.0000, A 0.000, B 0.000, C 0.000 }
gfCNCPoint5[29496] = {X 111.3156, Y 61.8692, Z -8.0000, A 0.000, B 0.000, C 0.000 }
gfCNCPoint5[29497] = {X 111.4013, Y 59.4708, Z -8.0000, A 0.000, B 0.000, C 0.000 }
gfCNCPoint5[29498] = {X 109.9149, Y 59.3407, Z -8.0000, A 0.000, B 0.000, C 0.000 }
gfCNCPoint5[29499] = {X 108.4496, Y 59.0584, Z -8.0000, A 0.000, B 0.000, C 0.000 }
gfCNCPoint5[29500] = {X 107.0213, Y 58.6267, Z -8.0000, A 0.000, B 0.000, C 0.000 }
gfCNCPoint5[29501] = {X 105.4260, Y 59.0985, Z -8.0000, A 0.000, B 0.000, C 0.000 }
gfCNCPoint5[29502] = {X 103.7872, Y 59.3842, Z -8.0000, A 0.000, B 0.000, C 0.000 }
gfCNCPoint5[29503] = {X 102.1264, Y 59.4800, Z -8.0000, A 0.000, B 0.000, C 0.000 }
gfCNCPoint5[29504] = {X 100.4656, Y 59.3847, Z -8.0000, A 0.000, B 0.000, C 0.000 }
gfCNCPoint5[29505] = {X 98.8267, Y 59.0996, Z -8.0000, A 0.000, B 0.000, C 0.000 }
gfCNCPoint5[29506] = {X 97.2313, Y 58.6283, Z -8.0000, A 0.000, B 0.000, C 0.000 }
gfCNCPoint5[29507] = {X 95.6367, Y 59.0994, Z -8.0000, A 0.000, B 0.000, C 0.000 }
gfCNCPoint5[29508] = {X 93.9986, Y 59.3845, Z -8.0000, A 0.000, B 0.000, C 0.000 }
gfCNCPoint5[29509] = {X 92.3385, Y 59.4800, Z -8.0000, A 0.000, B 0.000, C 0.000 }
gfCNCPoint5[29510] = {X 85.8951, Y 59.4800, Z -8.0000, A 0.000, B 0.000, C 0.000 }
gfCNCPoint5[29511] = {X 84.7780, Y 59.4368, Z -8.0000, A 0.000, B 0.000, C 0.000 }
gfCNCPoint5[29512] = {X 83.6677, Y 59.3077, Z -8.0000, A 0.000, B 0.000, C 0.000 }
gfCNCPoint5[29513] = {X 82.0978, Y 60.5827, Z -8.0000, A 0.000, B 0.000, C 0.000 }
gfCNCPoint5[29514] = {X 80.4031, Y 61.6862, Z -8.0000, A 0.000, B 0.000, C 0.000 }
gfCNCPoint5[29515] = {X 78.6021, Y 62.6061, Z -8.0000, A 0.000, B 0.000, C 0.000 }
gfCNCPoint5[29516] = {X 76.7146, Y 63.3324, Z -8.0000, A 0.000, B 0.000, C 0.000 }
gfCNCPoint5[29517] = {X 74.7614, Y 63.8569, Z -8.0000, A 0.000, B 0.000, C 0.000 }
gfCNCPoint5[29518] = {X 72.7640, Y 64.1739, Z -8.0000, A 0.000, B 0.000, C 0.000 }
gfCNCPoint5[29519] = {X 70.7445, Y 64.2800, Z -8.0000, A 0.000, B 0.000, C 0.000 }
gfCNCPoint5[29520] = {X 64.1851, Y 64.2800, Z -8.0000, A 0.000, B 0.000, C 0.000 }
gfCNCPoint5[29521] = {X 62.0428, Y 64.1606, Z -8.0000, A 0.000, B 0.000, C 0.000 }
gfCNCPoint5[29522] = {X 59.9269, Y 63.8039, Z -8.0000, A 0.000, B 0.000, C 0.000 }
gfCNCPoint5[29523] = {X 57.8638, Y 63.2143, Z -8.0000, A 0.000, B 0.000, C 0.000 }
gfCNCPoint5[29524] = {X 55.8790, Y 62.3991, Z -8.0000, A 0.000, B 0.000, C 0.000 }
gfCNCPoint5[29525] = {X 53.8942, Y 63.2143, Z -8.0000, A 0.000, B 0.000, C 0.000 }
gfCNCPoint5[29526] = {X 51.8311, Y 63.8039, Z -8.0000, A 0.000, B 0.000, C 0.000 }
gfCNCPoint5[29527] = {X 49.7153, Y 64.1606, Z -8.0000, A 0.000, B 0.000, C 0.000 }
gfCNCPoint5[29528] = {X 47.5729, Y 64.2800, Z -8.0000, A 0.000, B 0.000, C 0.000 }
gfCNCPoint5[29529] = {X 40.6393, Y 64.2800, Z -8.0000, A 0.000, B 0.000, C 0.000 }
gfCNCPoint5[29530] = {X 39.1553, Y 64.2228, Z -8.0000, A 0.000, B 0.000, C 0.000 }
gfCNCPoint5[29531] = {X 37.6801, Y 64.0516, Z -8.0000, A 0.000, B 0.000, C 0.000 }
gfCNCPoint5[29532] = {X 36.2225, Y 63.7673, Z -8.0000, A 0.000, B 0.000, C 0.000 }
gfCNCPoint5[29533] = {X 34.1359, Y 64.5955, Z -8.0000, A 0.000, B 0.000, C 0.000 }
gfCNCPoint5[29534] = {X 31.9801, Y 65.2219, Z -8.0000, A 0.000, B 0.000, C 0.000 }
gfCNCPoint5[29535] = {X 29.7746, Y 65.6406, Z -8.0000, A 0.000, B 0.000, C 0.000 }
gfCNCPoint5[29536] = {X 27.7191, Y 66.4656, Z -8.0000, A 0.000, B 0.000, C 0.000 }
gfCNCPoint5[29537] = {X 25.6283, Y 67.1963, Z -8.0000, A 0.000, B 0.000, C 0.000 }
gfCNCPoint5[29538] = {X 23.4824, Y 67.8391, Z -8.0000, A 0.000, B 0.000, C 0.000 }
gfCNCPoint5[29539] = {X 21.3054, Y 68.3666, Z -8.0000, A 0.000, B 0.000, C 0.000 }
gfCNCPoint5[29540] = {X 19.1033, Y 68.7775, Z -8.0000, A 0.000, B 0.000, C 0.000 }
gfCNCPoint5[29541] = {X 19.1033, Y 80.8952, Z -8.0000, A 0.000, B 0.000, C 0.000 }
gfCNCPoint5[29542] = {X 110.5595, Y 80.8952, Z -8.0000, A 0.000, B 0.000, C 0.000 }
gfCNCPoint5[29543] = {X 112.3059, Y 79.4909, Z -8.0000, A 0.000, B 0.000, C 0.000 }
gfCNCPoint5[29544] = {X 114.1879, Y 78.2744, Z -8.0000, A 0.000, B 0.000, C 0.000 }
gfCNCPoint5[29545] = {X 116.1854, Y 77.2587, Z -8.0000, A 0.000, B 0.000, C 0.000 }
gfCNCPoint5[29546] = {X 118.2771, Y 76.4546, Z -8.0000, A 0.000, B 0.000, C 0.000 }
gfCNCPoint5[29547] = {X 133.9622, Y 59.2314, Z -8.0000, A 0.000, B 0.000, C 0.000 }
gfCNCPoint5[29548] = {X 132.7148, Y 58.3541, Z -8.0000, A 0.000, B 0.000, C 0.000 }
gfCNCPoint5[29549] = {X 131.5517, Y 57.3678, Z -8.0000, A 0.000, B 0.000, C 0.000 }
gfCNCPoint5[29550] = {X 130.4824, Y 56.2805, Z -8.0000, A 0.000, B 0.000, C 0.000 }
gfCNCPoint5[29551] = {X 129.6655, Y 55.2988, Z -8.0000, A 0.000, B 0.000, C 0.000 }
gfCNCPoint5[29552] = {X 128.9251, Y 54.2582, Z -8.0000, A 0.000, B 0.000, C 0.000 }
gfCNCPoint5[29553] = {X 128.0750, Y 55.1942, Z -8.0000, A 0.000, B 0.000, C 0.000 }
gfCNCPoint5[29554] = {X 127.1464, Y 56.0525, Z -8.0000, A 0.000, B 0.000, C 0.000 }
gfCNCPoint5[29555] = {X 125.7915, Y 57.0695, Z -8.0000, A 0.000, B 0.000, C 0.000 }
gfCNCPoint5[29556] = {X 124.3270, Y 57.9212, Z -8.0000, A 0.000, B 0.000, C 0.000 }
gfCNCPoint5[29557] = {X 122.7731, Y 58.5961, Z -8.0000, A 0.000, B 0.000, C 0.000 }
gfCNCPoint5[29558] = {X 121.1510, Y 59.0849, Z -8.0000, A 0.000, B 0.000, C 0.000 }
gfCNCPoint5[29559] = {X 119.4828, Y 59.3809, Z -8.0000, A 0.000, B 0.000, C 0.000 }
gfCNCPoint5[29560] = {X 117.7916, Y 59.4800, Z -8.0000, A 0.000, B 0.000, C 0.000 }
gfCNCPoint5[29561] = {X 111.9185, Y 59.4800, Z -8.0000, A 0.000, B 0.000, C 0.000 }
gfCNCPoint5[29562] = {X 111.6599, Y 59.4777, Z -8.0000, A 0.000, B 0.000, C 0.000 }
gfCNCPoint5[29563] = {X 111.4013, Y 59.4708, Z -8.0000, A 0.000, B 0.000, C 0.000 }
gfCNCPoint5[29564] = {X 111.4871, Y 57.0723, Z -8.0000, A 0.000, B 0.000, C 0.000 }
gfCNCPoint5[29565] = {X 109.9587, Y 56.9200, Z -8.0000, A 0.000, B 0.000, C 0.000 }
gfCNCPoint5[29566] = {X 108.4621, Y 56.5750, Z -8.0000, A 0.000, B 0.000, C 0.000 }
gfCNCPoint5[29567] = {X 107.0213, Y 56.0428, Z -8.0000, A 0.000, B 0.000, C 0.000 }
gfCNCPoint5[29568] = {X 105.4432, Y 56.6151, Z -8.0000, A 0.000, B 0.000, C 0.000 }
gfCNCPoint5[29569] = {X 103.8010, Y 56.9630, Z -8.0000, A 0.000, B 0.000, C 0.000 }
gfCNCPoint5[29570] = {X 102.1265, Y 57.0800, Z -8.0000, A 0.000, B 0.000, C 0.000 }
gfCNCPoint5[29571] = {X 100.4519, Y 56.9637, Z -8.0000, A 0.000, B 0.000, C 0.000 }
gfCNCPoint5[29572] = {X 98.8096, Y 56.6164, Z -8.0000, A 0.000, B 0.000, C 0.000 }
gfCNCPoint5[29573] = {X 97.2313, Y 56.0448, Z -8.0000, A 0.000, B 0.000, C 0.000 }
gfCNCPoint5[29574] = {X 95.6538, Y 56.6162, Z -8.0000, A 0.000, B 0.000, C 0.000 }
gfCNCPoint5[29575] = {X 94.0123, Y 56.9635, Z -8.0000, A 0.000, B 0.000, C 0.000 }
gfCNCPoint5[29576] = {X 92.3385, Y 57.0800, Z -8.0000, A 0.000, B 0.000, C 0.000 }
gfCNCPoint5[29577] = {X 85.8951, Y 57.0800, Z -8.0000, A 0.000, B 0.000, C 0.000 }
gfCNCPoint5[29578] = {X 84.3894, Y 56.9858, Z -8.0000, A 0.000, B 0.000, C 0.000 }
gfCNCPoint5[29579] = {X 82.9073, Y 56.7047, Z -8.0000, A 0.000, B 0.000, C 0.000 }
gfCNCPoint5[29580] = {X 81.4847, Y 58.0224, Z -8.0000, A 0.000, B 0.000, C 0.000 }
gfCNCPoint5[29581] = {X 79.9203, Y 59.1682, Z -8.0000, A 0.000, B 0.000, C 0.000 }
gfCNCPoint5[29582] = {X 78.2348, Y 60.1271, Z -8.0000, A 0.000, B 0.000, C 0.000 }
gfCNCPoint5[29583] = {X 76.4504, Y 60.8864, Z -8.0000, A 0.000, B 0.000, C 0.000 }
gfCNCPoint5[29584] = {X 74.5908, Y 61.4359, Z -8.0000, A 0.000, B 0.000, C 0.000 }
gfCNCPoint5[29585] = {X 72.6804, Y 61.7686, Z -8.0000, A 0.000, B 0.000, C 0.000 }
gfCNCPoint5[29586] = {X 70.7445, Y 61.8800, Z -8.0000, A 0.000, B 0.000, C 0.000 }
gfCNCPoint5[29587] = {X 64.1851, Y 61.8800, Z -8.0000, A 0.000, B 0.000, C 0.000 }
gfCNCPoint5[29588] = {X 62.4514, Y 61.7907, Z -8.0000, A 0.000, B 0.000, C 0.000 }
gfCNCPoint5[29589] = {X 60.7359, Y 61.5238, Z -8.0000, A 0.000, B 0.000, C 0.000 }
gfCNCPoint5[29590] = {X 59.0570, Y 61.0822, Z -8.0000, A 0.000, B 0.000, C 0.000 }
gfCNCPoint5[29591] = {X 57.4323, Y 60.4704, Z -8.0000, A 0.000, B 0.000, C 0.000 }
gfCNCPoint5[29592] = {X 55.8790, Y 59.6950, Z -8.0000, A 0.000, B 0.000, C 0.000 }
gfCNCPoint5[29593] = {X 54.3258, Y 60.4704, Z -8.0000, A 0.000, B 0.000, C 0.000 }
gfCNCPoint5[29594] = {X 52.7011, Y 61.0822, Z -8.0000, A 0.000, B 0.000, C 0.000 }
gfCNCPoint5[29595] = {X 51.0221, Y 61.5238, Z -8.0000, A 0.000, B 0.000, C 0.000 }
gfCNCPoint5[29596] = {X 49.3067, Y 61.7907, Z -8.0000, A 0.000, B 0.000, C 0.000 }
gfCNCPoint5[29597] = {X 47.5729, Y 61.8800, Z -8.0000, A 0.000, B 0.000, C 0.000 }
gfCNCPoint5[29598] = {X 40.6393, Y 61.8800, Z -8.0000, A 0.000, B 0.000, C 0.000 }
gfCNCPoint5[29599] = {X 39.0682, Y 61.8067, Z -8.0000, A 0.000, B 0.000, C 0.000 }
gfCNCPoint5[29600] = {X 37.5107, Y 61.5875, Z -8.0000, A 0.000, B 0.000, C 0.000 }
gfCNCPoint5[29601] = {X 35.9804, Y 61.2243, Z -8.0000, A 0.000, B 0.000, C 0.000 }
gfCNCPoint5[29602] = {X 34.3397, Y 61.9612, Z -8.0000, A 0.000, B 0.000, C 0.000 }
gfCNCPoint5[29603] = {X 32.6424, Y 62.5564, Z -8.0000, A 0.000, B 0.000, C 0.000 }
gfCNCPoint5[29604] = {X 30.9008, Y 63.0056, Z -8.0000, A 0.000, B 0.000, C 0.000 }
gfCNCPoint5[29605] = {X 29.1275, Y 63.3057, Z -8.0000, A 0.000, B 0.000, C 0.000 }
gfCNCPoint5[29606] = {X 27.0252, Y 64.1623, Z -8.0000, A 0.000, B 0.000, C 0.000 }
gfCNCPoint5[29607] = {X 24.8834, Y 64.9148, Z -8.0000, A 0.000, B 0.000, C 0.000 }
gfCNCPoint5[29608] = {X 22.2004, Y 65.6938, Z -8.0000, A 0.000, B 0.000, C 0.000 }
gfCNCPoint5[29609] = {X 19.4692, Y 66.2818, Z -8.0000, A 0.000, B 0.000, C 0.000 }
gfCNCPoint5[29610] = {X 16.7033, Y 66.6760, Z -8.0000, A 0.000, B 0.000, C 0.000 }
gfCNCPoint5[29611] = {X 16.7033, Y 83.2952, Z -8.0000, A 0.000, B 0.000, C 0.000 }
gfCNCPoint5[29612] = {X 111.5061, Y 83.2952, Z -8.0000, A 0.000, B 0.000, C 0.000 }
gfCNCPoint5[29613] = {X 112.9241, Y 82.0362, Z -8.0000, A 0.000, B 0.000, C 0.000 }
gfCNCPoint5[29614] = {X 114.4589, Y 80.9227, Z -8.0000, A 0.000, B 0.000, C 0.000 }
gfCNCPoint5[29615] = {X 116.0957, Y 79.9653, Z -8.0000, A 0.000, B 0.000, C 0.000 }
gfCNCPoint5[29616] = {X 117.8186, Y 79.1733, Z -8.0000, A 0.000, B 0.000, C 0.000 }
gfCNCPoint5[29617] = {X 119.6110, Y 78.5544, Z -8.0000, A 0.000, B 0.000, C 0.000 }
gfCNCPoint5[29618] = {X 137.8559, Y 58.5203, Z -8.0000, A 0.000, B 0.000, C 0.000 }
gfCNCPoint5[29619] = {X 136.5212, Y 57.9298, Z -8.0000, A 0.000, B 0.000, C 0.000 }
gfCNCPoint5[29620] = {X 135.2528, Y 57.2080, Z -8.0000, A 0.000, B 0.000, C 0.000 }
gfCNCPoint5[29621] = {X 134.0092, Y 56.3191, Z -8.0000, A 0.000, B 0.000, C 0.000 }
gfCNCPoint5[29622] = {X 132.8662, Y 55.3040, Z -8.0000, A 0.000, B 0.000, C 0.000 }
gfCNCPoint5[29623] = {X 131.8366, Y 54.1741, Z -8.0000, A 0.000, B 0.000, C 0.000 }
gfCNCPoint5[29624] = {X 130.9319, Y 52.9419, Z -8.0000, A 0.000, B 0.000, C 0.000 }
gfCNCPoint5[29625] = {X 130.2147, Y 51.7225, Z -8.0000, A 0.000, B 0.000, C 0.000 }
gfCNCPoint5[29626] = {X 129.6199, Y 50.4390, Z -8.0000, A 0.000, B 0.000, C 0.000 }
gfCNCPoint5[29627] = {X 129.1532, Y 49.1035, Z -8.0000, A 0.000, B 0.000, C 0.000 }
gfCNCPoint5[29628] = {X 128.6036, Y 50.3877, Z -8.0000, A 0.000, B 0.000, C 0.000 }
gfCNCPoint5[29629] = {X 127.9093, Y 51.5998, Z -8.0000, A 0.000, B 0.000, C 0.000 }
gfCNCPoint5[29630] = {X 127.0798, Y 52.7237, Z -8.0000, A 0.000, B 0.000, C 0.000 }
gfCNCPoint5[29631] = {X 126.0417, Y 53.8239, Z -8.0000, A 0.000, B 0.000, C 0.000 }
gfCNCPoint5[29632] = {X 124.8743, Y 54.7858, Z -8.0000, A 0.000, B 0.000, C 0.000 }
gfCNCPoint5[29633] = {X 123.5958, Y 55.5942, Z -8.0000, A 0.000, B 0.000, C 0.000 }
gfCNCPoint5[29634] = {X 122.2263, Y 56.2365, Z -8.0000, A 0.000, B 0.000, C 0.000 }
gfCNCPoint5[29635] = {X 120.7872, Y 56.7027, Z -8.0000, A 0.000, B 0.000, C 0.000 }
gfCNCPoint5[29636] = {X 119.3012, Y 56.9853, Z -8.0000, A 0.000, B 0.000, C 0.000 }
gfCNCPoint5[29637] = {X 117.7916, Y 57.0800, Z -8.0000, A 0.000, B 0.000, C 0.000 }
gfCNCPoint5[29638] = {X 111.9185, Y 57.0800, Z -8.0000, A 0.000, B 0.000, C 0.000 }
gfCNCPoint5[29639] = {X 111.7027, Y 57.0781, Z -8.0000, A 0.000, B 0.000, C 0.000 }
gfCNCPoint5[29640] = {X 111.4871, Y 57.0723, Z -8.0000, A 0.000, B 0.000, C 0.000 }
gfCNCPoint5[29641] = {X 111.5728, Y 54.6738, Z -8.0000, A 0.000, B 0.000, C 0.000 }
gfCNCPoint5[29642] = {X 110.3820, Y 54.5573, Z -8.0000, A 0.000, B 0.000, C 0.000 }
gfCNCPoint5[29643] = {X 109.2147, Y 54.2947, Z -8.0000, A 0.000, B 0.000, C 0.000 }
gfCNCPoint5[29644] = {X 108.0887, Y 53.8902, Z -8.0000, A 0.000, B 0.000, C 0.000 }
gfCNCPoint5[29645] = {X 107.0213, Y 53.3498, Z -8.0000, A 0.000, B 0.000, C 0.000 }
gfCNCPoint5[29646] = {X 106.6480, Y 53.5578, Z -8.0000, A 0.000, B 0.000, C 0.000 }
gfCNCPoint5[29647] = {X 106.2658, Y 53.7492, Z -8.0000, A 0.000, B 0.000, C 0.000 }
gfCNCPoint5[29648] = {X 105.0149, Y 54.2383, Z -8.0000, A 0.000, B 0.000, C 0.000 }
gfCNCPoint5[29649] = {X 103.7084, Y 54.5495, Z -8.0000, A 0.000, B 0.000, C 0.000 }
gfCNCPoint5[29650] = {X 102.3713, Y 54.6768, Z -8.0000, A 0.000, B 0.000, C 0.000 }
gfCNCPoint5[29651] = {X 101.0295, Y 54.6179, Z -8.0000, A 0.000, B 0.000, C 0.000 }
gfCNCPoint5[29652] = {X 99.7088, Y 54.3738, Z -8.0000, A 0.000, B 0.000, C 0.000 }
gfCNCPoint5[29653] = {X 98.4345, Y 53.9493, Z -8.0000, A 0.000, B 0.000, C 0.000 }
gfCNCPoint5[29654] = {X 97.2313, Y 53.3524, Z -8.0000, A 0.000, B 0.000, C 0.000 }
gfCNCPoint5[29655] = {X 96.0852, Y 53.9255, Z -8.0000, A 0.000, B 0.000, C 0.000 }
gfCNCPoint5[29656] = {X 94.8734, Y 54.3422, Z -8.0000, A 0.000, B 0.000, C 0.000 }
gfCNCPoint5[29657] = {X 93.6172, Y 54.5952, Z -8.0000, A 0.000, B 0.000, C 0.000 }
gfCNCPoint5[29658] = {X 92.3385, Y 54.6800, Z -8.0000, A 0.000, B 0.000, C 0.000 }
gfCNCPoint5[29659] = {X 85.8951, Y 54.6800, Z -8.0000, A 0.000, B 0.000, C 0.000 }
gfCNCPoint5[29660] = {X 84.6159, Y 54.5951, Z -8.0000, A 0.000, B 0.000, C 0.000 }
gfCNCPoint5[29661] = {X 83.3592, Y 54.3419, Z -8.0000, A 0.000, B 0.000, C 0.000 }
gfCNCPoint5[29662] = {X 82.1469, Y 53.9249, Z -8.0000, A 0.000, B 0.000, C 0.000 }
gfCNCPoint5[29663] = {X 81.0644, Y 55.1572, Z -8.0000, A 0.000, B 0.000, C 0.000 }
gfCNCPoint5[29664] = {X 79.8495, Y 56.2591, Z -8.0000, A 0.000, B 0.000, C 0.000 }
gfCNCPoint5[29665] = {X 78.5178, Y 57.2166, Z -8.0000, A 0.000, B 0.000, C 0.000 }
gfCNCPoint5[29666] = {X 77.0863, Y 58.0174, Z -8.0000, A 0.000, B 0.000, C 0.000 }
gfCNCPoint5[29667] = {X 75.5734, Y 58.6511, Z -8.0000, A 0.000, B 0.000, C 0.000 }
gfCNCPoint5[29668] = {X 73.9986, Y 59.1096, Z -8.0000, A 0.000, B 0.000, C 0.000 }
gfCNCPoint5[29669] = {X 72.3820, Y 59.3871, Z -8.0000, A 0.000, B 0.000, C 0.000 }
gfCNCPoint5[29670] = {X 70.7445, Y 59.4800, Z -8.0000, A 0.000, B 0.000, C 0.000 }
gfCNCPoint5[29671] = {X 64.1851, Y 59.4800, Z -8.0000, A 0.000, B 0.000, C 0.000 }
gfCNCPoint5[29672] = {X 62.4203, Y 59.3720, Z -8.0000, A 0.000, B 0.000, C 0.000 }
gfCNCPoint5[29673] = {X 60.6818, Y 59.0498, Z -8.0000, A 0.000, B 0.000, C 0.000 }
gfCNCPoint5[29674] = {X 58.9955, Y 58.5181, Z -8.0000, A 0.000, B 0.000, C 0.000 }
gfCNCPoint5[29675] = {X 57.3866, Y 57.7848, Z -8.0000, A 0.000, B 0.000, C 0.000 }
gfCNCPoint5[29676] = {X 55.8790, Y 56.8608, Z -8.0000, A 0.000, B 0.000, C 0.000 }
gfCNCPoint5[29677] = {X 54.3715, Y 57.7848, Z -8.0000, A 0.000, B 0.000, C 0.000 }
gfCNCPoint5[29678] = {X 52.7626, Y 58.5181, Z -8.0000, A 0.000, B 0.000, C 0.000 }
gfCNCPoint5[29679] = {X 51.0763, Y 59.0498, Z -8.0000, A 0.000, B 0.000, C 0.000 }
gfCNCPoint5[29680] = {X 49.3378, Y 59.3720, Z -8.0000, A 0.000, B 0.000, C 0.000 }
gfCNCPoint5[29681] = {X 47.5729, Y 59.4800, Z -8.0000, A 0.000, B 0.000, C 0.000 }
gfCNCPoint5[29682] = {X 40.6393, Y 59.4800, Z -8.0000, A 0.000, B 0.000, C 0.000 }
gfCNCPoint5[29683] = {X 38.9799, Y 59.3846, Z -8.0000, A 0.000, B 0.000, C 0.000 }
gfCNCPoint5[29684] = {X 37.3424, Y 59.0997, Z -8.0000, A 0.000, B 0.000, C 0.000 }
gfCNCPoint5[29685] = {X 35.7484, Y 58.6290, Z -8.0000, A 0.000, B 0.000, C 0.000 }
gfCNCPoint5[29686] = {X 34.0328, Y 59.4882, Z -8.0000, A 0.000, B 0.000, C 0.000 }
gfCNCPoint5[29687] = {X 32.2386, Y 60.1682, Z -8.0000, A 0.000, B 0.000, C 0.000 }
gfCNCPoint5[29688] = {X 30.3844, Y 60.6618, Z -8.0000, A 0.000, B 0.000, C 0.000 }
gfCNCPoint5[29689] = {X 28.4897, Y 60.9640, Z -8.0000, A 0.000, B 0.000, C 0.000 }
gfCNCPoint5[29690] = {X 26.3362, Y 61.8564, Z -8.0000, A 0.000, B 0.000, C 0.000 }
gfCNCPoint5[29691] = {X 24.1385, Y 62.6333, Z -8.0000, A 0.000, B 0.000, C 0.000 }
gfCNCPoint5[29692] = {X 21.7314, Y 63.3367, Z -8.0000, A 0.000, B 0.000, C 0.000 }
gfCNCPoint5[29693] = {X 19.2824, Y 63.8764, Z -8.0000, A 0.000, B 0.000, C 0.000 }
gfCNCPoint5[29694] = {X 16.8026, Y 64.2500, Z -8.0000, A 0.000, B 0.000, C 0.000 }
gfCNCPoint5[29695] = {X 14.3033, Y 64.4559, Z -8.0000, A 0.000, B 0.000, C 0.000 }
gfCNCPoint5[29696] = {X 14.3033, Y 85.6952, Z -8.0000, A 0.000, B 0.000, C 0.000 }
gfCNCPoint5[29697] = {X 112.5244, Y 85.6952, Z -8.0000, A 0.000, B 0.000, C 0.000 }
gfCNCPoint5[29698] = {X 113.9427, Y 84.3117, Z -8.0000, A 0.000, B 0.000, C 0.000 }
gfCNCPoint5[29699] = {X 115.5133, Y 83.1039, Z -8.0000, A 0.000, B 0.000, C 0.000 }
gfCNCPoint5[29700] = {X 117.2146, Y 82.0885, Z -8.0000, A 0.000, B 0.000, C 0.000 }
gfCNCPoint5[29701] = {X 119.0232, Y 81.2795, Z -8.0000, A 0.000, B 0.000, C 0.000 }
gfCNCPoint5[29702] = {X 120.9141, Y 80.6879, Z -8.0000, A 0.000, B 0.000, C 0.000 }
gfCNCPoint5[29703] = {X 142.4278, Y 57.0645, Z -8.0000, A 0.000, B 0.000, C 0.000 }
gfCNCPoint5[29704] = {X 141.1649, Y 56.9336, Z -8.0000, A 0.000, B 0.000, C 0.000 }
gfCNCPoint5[29705] = {X 139.9228, Y 56.6710, Z -8.0000, A 0.000, B 0.000, C 0.000 }
gfCNCPoint5[29706] = {X 138.7151, Y 56.2794, Z -8.0000, A 0.000, B 0.000, C 0.000 }
gfCNCPoint5[29707] = {X 137.2782, Y 55.6176, Z -8.0000, A 0.000, B 0.000, C 0.000 }
gfCNCPoint5[29708] = {X 135.9402, Y 54.7736, Z -8.0000, A 0.000, B 0.000, C 0.000 }
gfCNCPoint5[29709] = {X 134.7239, Y 53.7621, Z -8.0000, A 0.000, B 0.000, C 0.000 }
gfCNCPoint5[29710] = {X 133.6502, Y 52.6003, Z -8.0000, A 0.000, B 0.000, C 0.000 }
gfCNCPoint5[29711] = {X 132.7375, Y 51.3082, Z -8.0000, A 0.000, B 0.000, C 0.000 }
gfCNCPoint5[29712] = {X 132.0015, Y 49.9079, Z -8.0000, A 0.000, B 0.000, C 0.000 }
gfCNCPoint5[29713] = {X 131.4549, Y 48.4234, Z -8.0000, A 0.000, B 0.000, C 0.000 }
gfCNCPoint5[29714] = {X 131.1845, Y 47.3200, Z -8.0000, A 0.000, B 0.000, C 0.000 }
gfCNCPoint5[29715] = {X 131.0190, Y 46.1961, Z -8.0000, A 0.000, B 0.000, C 0.000 }
gfCNCPoint5[29716] = {X 130.9598, Y 45.0616, Z -8.0000, A 0.000, B 0.000, C 0.000 }
gfCNCPoint5[29717] = {X 130.9601, Y 44.0979, Z -8.0000, A 0.000, B 0.000, C 0.000 }
gfCNCPoint5[29718] = {X 131.0921, Y 42.4244, Z -8.0000, A 0.000, B 0.000, C 0.000 }
gfCNCPoint5[29719] = {X 131.4548, Y 40.7854, Z -8.0000, A 0.000, B 0.000, C 0.000 }
gfCNCPoint5[29720] = {X 133.7565, Y 41.4655, Z -8.0000, A 0.000, B 0.000, C 0.000 }
gfCNCPoint5[29721] = {X 134.2330, Y 40.1906, Z -8.0000, A 0.000, B 0.000, C 0.000 }
gfCNCPoint5[29722] = {X 134.8836, Y 38.9952, Z -8.0000, A 0.000, B 0.000, C 0.000 }
gfCNCPoint5[29723] = {X 134.8836, Y 27.0854, Z -8.0000, A 0.000, B 0.000, C 0.000 }
gfCNCPoint5[29724] = {X 134.3931, Y 27.1259, Z -8.0000, A 0.000, B 0.000, C 0.000 }
gfCNCPoint5[29725] = {X 133.9011, Y 27.1414, Z -8.0000, A 0.000, B 0.000, C 0.000 }
gfCNCPoint5[29726] = {X 133.2006, Y 27.1415, Z -8.0000, A 0.000, B 0.000, C 0.000 }
gfCNCPoint5[29727] = {X 131.9568, Y 27.0613, Z -8.0000, A 0.000, B 0.000, C 0.000 }
gfCNCPoint5[29728] = {X 130.7335, Y 26.8219, Z -8.0000, A 0.000, B 0.000, C 0.000 }
gfCNCPoint5[29729] = {X 129.5512, Y 26.4273, Z -8.0000, A 0.000, B 0.000, C 0.000 }
gfCNCPoint5[29730] = {X 128.4294, Y 25.8840, Z -8.0000, A 0.000, B 0.000, C 0.000 }
gfCNCPoint5[29731] = {X 127.3867, Y 25.2011, Z -8.0000, A 0.000, B 0.000, C 0.000 }
gfCNCPoint5[29732] = {X 126.3461, Y 24.2965, Z -8.0000, A 0.000, B 0.000, C 0.000 }
gfCNCPoint5[29733] = {X 125.4445, Y 23.2533, Z -8.0000, A 0.000, B 0.000, C 0.000 }
gfCNCPoint5[29734] = {X 124.7003, Y 22.0926, Z -8.0000, A 0.000, B 0.000, C 0.000 }
gfCNCPoint5[29735] = {X 124.1286, Y 20.8380, Z -8.0000, A 0.000, B 0.000, C 0.000 }
gfCNCPoint5[29736] = {X 123.7409, Y 19.5148, Z -8.0000, A 0.000, B 0.000, C 0.000 }
gfCNCPoint5[29737] = {X 123.5452, Y 18.1500, Z -8.0000, A 0.000, B 0.000, C 0.000 }
gfCNCPoint5[29738] = {X 123.5453, Y 39.7486, Z -8.0000, A 0.000, B 0.000, C 0.000 }
gfCNCPoint5[29739] = {X 124.1933, Y 40.7423, Z -8.0000, A 0.000, B 0.000, C 0.000 }
gfCNCPoint5[29740] = {X 124.6713, Y 41.8280, Z -8.0000, A 0.000, B 0.000, C 0.000 }
gfCNCPoint5[29741] = {X 124.9666, Y 42.9770, Z -8.0000, A 0.000, B 0.000, C 0.000 }
gfCNCPoint5[29742] = {X 125.0714, Y 44.1587, Z -8.0000, A 0.000, B 0.000, C 0.000 }
gfCNCPoint5[29743] = {X 125.0716, Y 45.0000, Z -8.0000, A 0.000, B 0.000, C 0.000 }
gfCNCPoint5[29744] = {X 124.9610, Y 46.2642, Z -8.0000, A 0.000, B 0.000, C 0.000 }
gfCNCPoint5[29745] = {X 124.6325, Y 47.4899, Z -8.0000, A 0.000, B 0.000, C 0.000 }
gfCNCPoint5[29746] = {X 124.0962, Y 48.6400, Z -8.0000, A 0.000, B 0.000, C 0.000 }
gfCNCPoint5[29747] = {X 123.3684, Y 49.6795, Z -8.0000, A 0.000, B 0.000, C 0.000 }
gfCNCPoint5[29748] = {X 122.4711, Y 50.5768, Z -8.0000, A 0.000, B 0.000, C 0.000 }
gfCNCPoint5[29749] = {X 121.4316, Y 51.3047, Z -8.0000, A 0.000, B 0.000, C 0.000 }
gfCNCPoint5[29750] = {X 120.2815, Y 51.8410, Z -8.0000, A 0.000, B 0.000, C 0.000 }
gfCNCPoint5[29751] = {X 119.0557, Y 52.1694, Z -8.0000, A 0.000, B 0.000, C 0.000 }
gfCNCPoint5[29752] = {X 117.7916, Y 52.2800, Z -8.0000, A 0.000, B 0.000, C 0.000 }
gfCNCPoint5[29753] = {X 111.9185, Y 52.2800, Z -8.0000, A 0.000, B 0.000, C 0.000 }
gfCNCPoint5[29754] = {X 110.8481, Y 52.2009, Z -8.0000, A 0.000, B 0.000, C 0.000 }
gfCNCPoint5[29755] = {X 109.8009, Y 51.9652, Z -8.0000, A 0.000, B 0.000, C 0.000 }
gfCNCPoint5[29756] = {X 108.7998, Y 51.5782, Z -8.0000, A 0.000, B 0.000, C 0.000 }
gfCNCPoint5[29757] = {X 107.8665, Y 51.0481, Z -8.0000, A 0.000, B 0.000, C 0.000 }
gfCNCPoint5[29758] = {X 107.0213, Y 50.3866, Z -8.0000, A 0.000, B 0.000, C 0.000 }
gfCNCPoint5[29759] = {X 106.1743, Y 51.0493, Z -8.0000, A 0.000, B 0.000, C 0.000 }
gfCNCPoint5[29760] = {X 105.2389, Y 51.5800, Z -8.0000, A 0.000, B 0.000, C 0.000 }
gfCNCPoint5[29761] = {X 104.0917, Y 52.0091, Z -8.0000, A 0.000, B 0.000, C 0.000 }
gfCNCPoint5[29762] = {X 102.8887, Y 52.2397, Z -8.0000, A 0.000, B 0.000, C 0.000 }
gfCNCPoint5[29763] = {X 101.6641, Y 52.2655, Z -8.0000, A 0.000, B 0.000, C 0.000 }
gfCNCPoint5[29764] = {X 100.4526, Y 52.0855, Z -8.0000, A 0.000, B 0.000, C 0.000 }
gfCNCPoint5[29765] = {X 99.2883, Y 51.7050, Z -8.0000, A 0.000, B 0.000, C 0.000 }
gfCNCPoint5[29766] = {X 98.2043, Y 51.1347, Z -8.0000, A 0.000, B 0.000, C 0.000 }
gfCNCPoint5[29767] = {X 97.2313, Y 50.3907, Z -8.0000, A 0.000, B 0.000, C 0.000 }
gfCNCPoint5[29768] = {X 96.3865, Y 51.0508, Z -8.0000, A 0.000, B 0.000, C 0.000 }
gfCNCPoint5[29769] = {X 95.4539, Y 51.5797, Z -8.0000, A 0.000, B 0.000, C 0.000 }
gfCNCPoint5[29770] = {X 94.4538, Y 51.9659, Z -8.0000, A 0.000, B 0.000, C 0.000 }
gfCNCPoint5[29771] = {X 93.4078, Y 52.2011, Z -8.0000, A 0.000, B 0.000, C 0.000 }
gfCNCPoint5[29772] = {X 92.3385, Y 52.2800, Z -8.0000, A 0.000, B 0.000, C 0.000 }
gfCNCPoint5[29773] = {X 85.8951, Y 52.2800, Z -8.0000, A 0.000, B 0.000, C 0.000 }
gfCNCPoint5[29774] = {X 84.6852, Y 52.1788, Z -8.0000, A 0.000, B 0.000, C 0.000 }
gfCNCPoint5[29775] = {X 83.5090, Y 51.8779, Z -8.0000, A 0.000, B 0.000, C 0.000 }
gfCNCPoint5[29776] = {X 82.3992, Y 51.3857, Z -8.0000, A 0.000, B 0.000, C 0.000 }
gfCNCPoint5[29777] = {X 81.3866, Y 50.7159, Z -8.0000, A 0.000, B 0.000, C 0.000 }
gfCNCPoint5[29778] = {X 80.5223, Y 52.0937, Z -8.0000, A 0.000, B 0.000, C 0.000 }
gfCNCPoint5[29779] = {X 79.4808, Y 53.3429, Z -8.0000, A 0.000, B 0.000, C 0.000 }
gfCNCPoint5[29780] = {X 78.2809, Y 54.4408, Z -8.0000, A 0.000, B 0.000, C 0.000 }
gfCNCPoint5[29781] = {X 76.9444, Y 55.3676, Z -8.0000, A 0.000, B 0.000, C 0.000 }
gfCNCPoint5[29782] = {X 75.4955, Y 56.1065, Z -8.0000, A 0.000, B 0.000, C 0.000 }
gfCNCPoint5[29783] = {X 73.9605, Y 56.6440, Z -8.0000, A 0.000, B 0.000, C 0.000 }
gfCNCPoint5[29784] = {X 72.3672, Y 56.9705, Z -8.0000, A 0.000, B 0.000, C 0.000 }
gfCNCPoint5[29785] = {X 70.7445, Y 57.0800, Z -8.0000, A 0.000, B 0.000, C 0.000 }
gfCNCPoint5[29786] = {X 64.1851, Y 57.0800, Z -8.0000, A 0.000, B 0.000, C 0.000 }
gfCNCPoint5[29787] = {X 62.6628, Y 56.9837, Z -8.0000, A 0.000, B 0.000, C 0.000 }
gfCNCPoint5[29788] = {X 61.1646, Y 56.6963, Z -8.0000, A 0.000, B 0.000, C 0.000 }
gfCNCPoint5[29789] = {X 59.7147, Y 56.2224, Z -8.0000, A 0.000, B 0.000, C 0.000 }
gfCNCPoint5[29790] = {X 58.3360, Y 55.5695, Z -8.0000, A 0.000, B 0.000, C 0.000 }
gfCNCPoint5[29791] = {X 57.0507, Y 54.7481, Z -8.0000, A 0.000, B 0.000, C 0.000 }
gfCNCPoint5[29792] = {X 55.8790, Y 53.7713, Z -8.0000, A 0.000, B 0.000, C 0.000 }
gfCNCPoint5[29793] = {X 54.7074, Y 54.7481, Z -8.0000, A 0.000, B 0.000, C 0.000 }
gfCNCPoint5[29794] = {X 53.4220, Y 55.5695, Z -8.0000, A 0.000, B 0.000, C 0.000 }
gfCNCPoint5[29795] = {X 52.0434, Y 56.2224, Z -8.0000, A 0.000, B 0.000, C 0.000 }
gfCNCPoint5[29796] = {X 50.5934, Y 56.6963, Z -8.0000, A 0.000, B 0.000, C 0.000 }
gfCNCPoint5[29797] = {X 49.0953, Y 56.9837, Z -8.0000, A 0.000, B 0.000, C 0.000 }
gfCNCPoint5[29798] = {X 47.5729, Y 57.0800, Z -8.0000, A 0.000, B 0.000, C 0.000 }
gfCNCPoint5[29799] = {X 40.6393, Y 57.0800, Z -8.0000, A 0.000, B 0.000, C 0.000 }
gfCNCPoint5[29800] = {X 39.3239, Y 57.0082, Z -8.0000, A 0.000, B 0.000, C 0.000 }
gfCNCPoint5[29801] = {X 38.0241, Y 56.7935, Z -8.0000, A 0.000, B 0.000, C 0.000 }
gfCNCPoint5[29802] = {X 36.7554, Y 56.4386, Z -8.0000, A 0.000, B 0.000, C 0.000 }
gfCNCPoint5[29803] = {X 35.5330, Y 55.9477, Z -8.0000, A 0.000, B 0.000, C 0.000 }
gfCNCPoint5[29804] = {X 34.1216, Y 56.7832, Z -8.0000, A 0.000, B 0.000, C 0.000 }
gfCNCPoint5[29805] = {X 32.6338, Y 57.4736, Z -8.0000, A 0.000, B 0.000, C 0.000 }
gfCNCPoint5[29806] = {X 31.0846, Y 58.0121, Z -8.0000, A 0.000, B 0.000, C 0.000 }
gfCNCPoint5[29807] = {X 29.4894, Y 58.3932, Z -8.0000, A 0.000, B 0.000, C 0.000 }
gfCNCPoint5[29808] = {X 27.8640, Y 58.6132, Z -8.0000, A 0.000, B 0.000, C 0.000 }
gfCNCPoint5[29809] = {X 25.6539, Y 59.5472, Z -8.0000, A 0.000, B 0.000, C 0.000 }
gfCNCPoint5[29810] = {X 23.3935, Y 60.3519, Z -8.0000, A 0.000, B 0.000, C 0.000 }
gfCNCPoint5[29811] = {X 21.1527, Y 61.0074, Z -8.0000, A 0.000, B 0.000, C 0.000 }
gfCNCPoint5[29812] = {X 18.8729, Y 61.5114, Z -8.0000, A 0.000, B 0.000, C 0.000 }
gfCNCPoint5[29813] = {X 16.5645, Y 61.8615, Z -8.0000, A 0.000, B 0.000, C 0.000 }
gfCNCPoint5[29814] = {X 14.2378, Y 62.0562, Z -8.0000, A 0.000, B 0.000, C 0.000 }
gfCNCPoint5[29815] = {X 11.9033, Y 62.0946, Z -8.0000, A 0.000, B 0.000, C 0.000 }
gfCNCPoint5[29816] = {X 11.9033, Y 88.0952, Z -8.0000, A 0.000, B 0.000, C 0.000 }
gfCNCPoint5[29817] = {X 113.6336, Y 88.0952, Z -8.0000, A 0.000, B 0.000, C 0.000 }
gfCNCPoint5[29818] = {X 114.7663, Y 86.8218, Z -8.0000, A 0.000, B 0.000, C 0.000 }
gfCNCPoint5[29819] = {X 116.0408, Y 85.6904, Z -8.0000, A 0.000, B 0.000, C 0.000 }
gfCNCPoint5[29820] = {X 117.4393, Y 84.7166, Z -8.0000, A 0.000, B 0.000, C 0.000 }
gfCNCPoint5[29821] = {X 118.9426, Y 83.9138, Z -8.0000, A 0.000, B 0.000, C 0.000 }
gfCNCPoint5[29822] = {X 120.5299, Y 83.2932, Z -8.0000, A 0.000, B 0.000, C 0.000 }
gfCNCPoint5[29823] = {X 122.1790, Y 82.8634, Z -8.0000, A 0.000, B 0.000, C 0.000 }
gfCNCPoint5[29824] = {X 144.8180, Y 58.0043, Z -8.0000, A 0.000, B 0.000, C 0.000 }
gfCNCPoint5[29825] = {X 144.9145, Y 56.3310, Z -8.0000, A 0.000, B 0.000, C 0.000 }
gfCNCPoint5[29826] = {X 145.2037, Y 54.6800, Z -8.0000, A 0.000, B 0.000, C 0.000 }
gfCNCPoint5[29827] = {X 143.0396, Y 54.6800, Z -8.0000, A 0.000, B 0.000, C 0.000 }
gfCNCPoint5[29828] = {X 142.7944, Y 54.6769, Z -8.0000, A 0.000, B 0.000, C 0.000 }
gfCNCPoint5[29829] = {X 142.5493, Y 54.6676, Z -8.0000, A 0.000, B 0.000, C 0.000 }
gfCNCPoint5[29830] = {X 141.0965, Y 54.4830, Z -8.0000, A 0.000, B 0.000, C 0.000 }
gfCNCPoint5[29831] = {X 139.6881, Y 54.0813, Z -8.0000, A 0.000, B 0.000, C 0.000 }
gfCNCPoint5[29832] = {X 138.3564, Y 53.4717, Z -8.0000, A 0.000, B 0.000, C 0.000 }
gfCNCPoint5[29833] = {X 137.1319, Y 52.6682, Z -8.0000, A 0.000, B 0.000, C 0.000 }
gfCNCPoint5[29834] = {X 136.0427, Y 51.6892, Z -8.0000, A 0.000, B 0.000, C 0.000 }
gfCNCPoint5[29835] = {X 135.1136, Y 50.5570, Z -8.0000, A 0.000, B 0.000, C 0.000 }
gfCNCPoint5[29836] = {X 134.3660, Y 49.2977, Z -8.0000, A 0.000, B 0.000, C 0.000 }
gfCNCPoint5[29837] = {X 133.8169, Y 47.9399, Z -8.0000, A 0.000, B 0.000, C 0.000 }
gfCNCPoint5[29838] = {X 133.4789, Y 46.5149, Z -8.0000, A 0.000, B 0.000, C 0.000 }
gfCNCPoint5[29839] = {X 133.3598, Y 45.0552, Z -8.0000, A 0.000, B 0.000, C 0.000 }
gfCNCPoint5[29840] = {X 133.3601, Y 44.1105, Z -8.0000, A 0.000, B 0.000, C 0.000 }
gfCNCPoint5[29841] = {X 133.4665, Y 42.7743, Z -8.0000, A 0.000, B 0.000, C 0.000 }
gfCNCPoint5[29842] = {X 133.7565, Y 41.4655, Z -8.0000, A 0.000, B 0.000, C 0.000 }
gfCNCPoint5[29843] = {X 136.0581, Y 42.1457, Z -8.0000, A 0.000, B 0.000, C 0.000 }
gfCNCPoint5[29844] = {X 136.3664, Y 41.2990, Z -8.0000, A 0.000, B 0.000, C 0.000 }
gfCNCPoint5[29845] = {X 136.7770, Y 40.4969, Z -8.0000, A 0.000, B 0.000, C 0.000 }
gfCNCPoint5[29846] = {X 137.2836, Y 39.7516, Z -8.0000, A 0.000, B 0.000, C 0.000 }
gfCNCPoint5[29847] = {X 137.2836, Y 23.8768, Z -8.0000, A 0.000, B 0.000, C 0.000 }
gfCNCPoint5[29848] = {X 136.4352, Y 24.2641, Z -8.0000, A 0.000, B 0.000, C 0.000 }
gfCNCPoint5[29849] = {X 135.5443, Y 24.5398, Z -8.0000, A 0.000, B 0.000, C 0.000 }
gfCNCPoint5[29850] = {X 134.6254, Y 24.6993, Z -8.0000, A 0.000, B 0.000, C 0.000 }
gfCNCPoint5[29851] = {X 134.2595, Y 24.7296, Z -8.0000, A 0.000, B 0.000, C 0.000 }
gfCNCPoint5[29852] = {X 133.8926, Y 24.7414, Z -8.0000, A 0.000, B 0.000, C 0.000 }
gfCNCPoint5[29853] = {X 133.2006, Y 24.7415, Z -8.0000, A 0.000, B 0.000, C 0.000 }
gfCNCPoint5[29854] = {X 131.9932, Y 24.6407, Z -8.0000, A 0.000, B 0.000, C 0.000 }
gfCNCPoint5[29855] = {X 130.8193, Y 24.3410, Z -8.0000, A 0.000, B 0.000, C 0.000 }
gfCNCPoint5[29856] = {X 129.7113, Y 23.8508, Z -8.0000, A 0.000, B 0.000, C 0.000 }
gfCNCPoint5[29857] = {X 128.6999, Y 23.1836, Z -8.0000, A 0.000, B 0.000, C 0.000 }
gfCNCPoint5[29858] = {X 127.8132, Y 22.3579, Z -8.0000, A 0.000, B 0.000, C 0.000 }
gfCNCPoint5[29859] = {X 127.0758, Y 21.3965, Z -8.0000, A 0.000, B 0.000, C 0.000 }
gfCNCPoint5[29860] = {X 126.5079, Y 20.3262, Z -8.0000, A 0.000, B 0.000, C 0.000 }
gfCNCPoint5[29861] = {X 126.1255, Y 19.1765, Z -8.0000, A 0.000, B 0.000, C 0.000 }
gfCNCPoint5[29862] = {X 125.9391, Y 17.9793, Z -8.0000, A 0.000, B 0.000, C 0.000 }
gfCNCPoint5[29863] = {X 125.9253, Y 17.7206, Z -8.0000, A 0.000, B 0.000, C 0.000 }
gfCNCPoint5[29864] = {X 125.9206, Y 17.4615, Z -8.0000, A 0.000, B 0.000, C 0.000 }
gfCNCPoint5[29865] = {X 125.9206, Y 10.4835, Z -8.0000, A 0.000, B 0.000, C 0.000 }
gfCNCPoint5[29866] = {X 125.9372, Y 9.9931, Z -8.0000, A 0.000, B 0.000, C 0.000 }
gfCNCPoint5[29867] = {X 125.9867, Y 9.5048, Z -8.0000, A 0.000, B 0.000, C 0.000 }
gfCNCPoint5[29868] = {X 121.8685, Y 9.5048, Z -8.0000, A 0.000, B 0.000, C 0.000 }
gfCNCPoint5[29869] = {X 122.3090, Y 10.3409, Z -8.0000, A 0.000, B 0.000, C 0.000 }
gfCNCPoint5[29870] = {X 122.5801, Y 11.2462, Z -8.0000, A 0.000, B 0.000, C 0.000 }
gfCNCPoint5[29871] = {X 122.6716, Y 12.1868, Z -8.0000, A 0.000, B 0.000, C 0.000 }
gfCNCPoint5[29872] = {X 122.6714, Y 13.0237, Z -8.0000, A 0.000, B 0.000, C 0.000 }
gfCNCPoint5[29873] = {X 122.5640, Y 13.9968, Z -8.0000, A 0.000, B 0.000, C 0.000 }
gfCNCPoint5[29874] = {X 122.2647, Y 14.9289, Z -8.0000, A 0.000, B 0.000, C 0.000 }
gfCNCPoint5[29875] = {X 121.7853, Y 15.7824, Z -8.0000, A 0.000, B 0.000, C 0.000 }
gfCNCPoint5[29876] = {X 121.1452, Y 16.5231, Z -8.0000, A 0.000, B 0.000, C 0.000 }
gfCNCPoint5[29877] = {X 121.1453, Y 40.6638, Z -8.0000, A 0.000, B 0.000, C 0.000 }
gfCNCPoint5[29878] = {X 121.7862, Y 41.4056, Z -8.0000, A 0.000, B 0.000, C 0.000 }
gfCNCPoint5[29879] = {X 122.2658, Y 42.2606, Z -8.0000, A 0.000, B 0.000, C 0.000 }
gfCNCPoint5[29880] = {X 122.5649, Y 43.1942, Z -8.0000, A 0.000, B 0.000, C 0.000 }
gfCNCPoint5[29881] = {X 122.6714, Y 44.1688, Z -8.0000, A 0.000, B 0.000, C 0.000 }
gfCNCPoint5[29882] = {X 122.6716, Y 45.0000, Z -8.0000, A 0.000, B 0.000, C 0.000 }
gfCNCPoint5[29883] = {X 122.5778, Y 45.9520, Z -8.0000, A 0.000, B 0.000, C 0.000 }
gfCNCPoint5[29884] = {X 122.3001, Y 46.8675, Z -8.0000, A 0.000, B 0.000, C 0.000 }
gfCNCPoint5[29885] = {X 121.8491, Y 47.7112, Z -8.0000, A 0.000, B 0.000, C 0.000 }
gfCNCPoint5[29886] = {X 121.2423, Y 48.4507, Z -8.0000, A 0.000, B 0.000, C 0.000 }
gfCNCPoint5[29887] = {X 120.5028, Y 49.0576, Z -8.0000, A 0.000, B 0.000, C 0.000 }
gfCNCPoint5[29888] = {X 119.6591, Y 49.5085, Z -8.0000, A 0.000, B 0.000, C 0.000 }
gfCNCPoint5[29889] = {X 118.7436, Y 49.7862, Z -8.0000, A 0.000, B 0.000, C 0.000 }
gfCNCPoint5[29890] = {X 117.7916, Y 49.8800, Z -8.0000, A 0.000, B 0.000, C 0.000 }
gfCNCPoint5[29891] = {X 111.9185, Y 49.8800, Z -8.0000, A 0.000, B 0.000, C 0.000 }
gfCNCPoint5[29892] = {X 111.0234, Y 49.7972, Z -8.0000, A 0.000, B 0.000, C 0.000 }
gfCNCPoint5[29893] = {X 110.1587, Y 49.5517, Z -8.0000, A 0.000, B 0.000, C 0.000 }
gfCNCPoint5[29894] = {X 109.3537, Y 49.1517, Z -8.0000, A 0.000, B 0.000, C 0.000 }
gfCNCPoint5[29895] = {X 108.6357, Y 48.6108, Z -8.0000, A 0.000, B 0.000, C 0.000 }
gfCNCPoint5[29896] = {X 108.0714, Y 48.0024, Z -8.0000, A 0.000, B 0.000, C 0.000 }
gfCNCPoint5[29897] = {X 107.6183, Y 47.3071, Z -8.0000, A 0.000, B 0.000, C 0.000 }
gfCNCPoint5[29898] = {X 107.2895, Y 46.5451, Z -8.0000, A 0.000, B 0.000, C 0.000 }
gfCNCPoint5[29899] = {X 107.0947, Y 45.7384, Z -8.0000, A 0.000, B 0.000, C 0.000 }
gfCNCPoint5[29900] = {X 106.6287, Y 46.8769, Z -8.0000, A 0.000, B 0.000, C 0.000 }
gfCNCPoint5[29901] = {X 106.1131, Y 47.8110, Z -8.0000, A 0.000, B 0.000, C 0.000 }
gfCNCPoint5[29902] = {X 105.4068, Y 48.6108, Z -8.0000, A 0.000, B 0.000, C 0.000 }
gfCNCPoint5[29903] = {X 104.8391, Y 49.0550, Z -8.0000, A 0.000, B 0.000, C 0.000 }
gfCNCPoint5[29904] = {X 104.2121, Y 49.4107, Z -8.0000, A 0.000, B 0.000, C 0.000 }
gfCNCPoint5[29905] = {X 103.3106, Y 49.7335, Z -8.0000, A 0.000, B 0.000, C 0.000 }
gfCNCPoint5[29906] = {X 102.3635, Y 49.8741, Z -8.0000, A 0.000, B 0.000, C 0.000 }
gfCNCPoint5[29907] = {X 101.4071, Y 49.8271, Z -8.0000, A 0.000, B 0.000, C 0.000 }
gfCNCPoint5[29908] = {X 100.4784, Y 49.5941, Z -8.0000, A 0.000, B 0.000, C 0.000 }
gfCNCPoint5[29909] = {X 99.6130, Y 49.1844, Z -8.0000, A 0.000, B 0.000, C 0.000 }
gfCNCPoint5[29910] = {X 98.8443, Y 48.6135, Z -8.0000, A 0.000, B 0.000, C 0.000 }
gfCNCPoint5[29911] = {X 98.1362, Y 47.8127, Z -8.0000, A 0.000, B 0.000, C 0.000 }
gfCNCPoint5[29912] = {X 97.6194, Y 46.8769, Z -8.0000, A 0.000, B 0.000, C 0.000 }
gfCNCPoint5[29913] = {X 97.1600, Y 45.7536, Z -8.0000, A 0.000, B 0.000, C 0.000 }
gfCNCPoint5[29914] = {X 96.9635, Y 46.5570, Z -8.0000, A 0.000, B 0.000, C 0.000 }
gfCNCPoint5[29915] = {X 96.6342, Y 47.3156, Z -8.0000, A 0.000, B 0.000, C 0.000 }
gfCNCPoint5[29916] = {X 96.1814, Y 48.0078, Z -8.0000, A 0.000, B 0.000, C 0.000 }
gfCNCPoint5[29917] = {X 95.6183, Y 48.6135, Z -8.0000, A 0.000, B 0.000, C 0.000 }
gfCNCPoint5[29918] = {X 94.9007, Y 49.1533, Z -8.0000, A 0.000, B 0.000, C 0.000 }
gfCNCPoint5[29919] = {X 94.0964, Y 49.5524, Z -8.0000, A 0.000, B 0.000, C 0.000 }
gfCNCPoint5[29920] = {X 93.2326, Y 49.7974, Z -8.0000, A 0.000, B 0.000, C 0.000 }
gfCNCPoint5[29921] = {X 92.3385, Y 49.8800, Z -8.0000, A 0.000, B 0.000, C 0.000 }
gfCNCPoint5[29922] = {X 85.8951, Y 49.8800, Z -8.0000, A 0.000, B 0.000, C 0.000 }
gfCNCPoint5[29923] = {X 85.0841, Y 49.8121, Z -8.0000, A 0.000, B 0.000, C 0.000 }
gfCNCPoint5[29924] = {X 84.2956, Y 49.6104, Z -8.0000, A 0.000, B 0.000, C 0.000 }
gfCNCPoint5[29925] = {X 83.5517, Y 49.2805, Z -8.0000, A 0.000, B 0.000, C 0.000 }
gfCNCPoint5[29926] = {X 82.8729, Y 48.8316, Z -8.0000, A 0.000, B 0.000, C 0.000 }
gfCNCPoint5[29927] = {X 82.2391, Y 48.2324, Z -8.0000, A 0.000, B 0.000, C 0.000 }
gfCNCPoint5[29928] = {X 81.7221, Y 47.5300, Z -8.0000, A 0.000, B 0.000, C 0.000 }
gfCNCPoint5[29929] = {X 81.3384, Y 46.7467, Z -8.0000, A 0.000, B 0.000, C 0.000 }
gfCNCPoint5[29930] = {X 81.1002, Y 45.9077, Z -8.0000, A 0.000, B 0.000, C 0.000 }
gfCNCPoint5[29931] = {X 81.0152, Y 45.0397, Z -8.0000, A 0.000, B 0.000, C 0.000 }
gfCNCPoint5[29932] = {X 81.0151, Y 44.2046, Z -8.0000, A 0.000, B 0.000, C 0.000 }
gfCNCPoint5[29933] = {X 81.1190, Y 43.2205, Z -8.0000, A 0.000, B 0.000, C 0.000 }
gfCNCPoint5[29934] = {X 81.4173, Y 42.2770, Z -8.0000, A 0.000, B 0.000, C 0.000 }
gfCNCPoint5[29935] = {X 81.8980, Y 41.4119, Z -8.0000, A 0.000, B 0.000, C 0.000 }
gfCNCPoint5[29936] = {X 82.5416, Y 40.6602, Z -8.0000, A 0.000, B 0.000, C 0.000 }
gfCNCPoint5[29937] = {X 82.5416, Y 25.2445, Z -8.0000, A 0.000, B 0.000, C 0.000 }
gfCNCPoint5[29938] = {X 77.7416, Y 25.2445, Z -8.0000, A 0.000, B 0.000, C 0.000 }
gfCNCPoint5[29939] = {X 77.7417, Y 18.1957, Z -8.0000, A 0.000, B 0.000, C 0.000 }
gfCNCPoint5[29940] = {X 77.0776, Y 16.9724, Z -8.0000, A 0.000, B 0.000, C 0.000 }
gfCNCPoint5[29941] = {X 76.5959, Y 15.6664, Z -8.0000, A 0.000, B 0.000, C 0.000 }
gfCNCPoint5[29942] = {X 76.3064, Y 14.3048, Z -8.0000, A 0.000, B 0.000, C 0.000 }
gfCNCPoint5[29943] = {X 74.0412, Y 14.3048, Z -8.0000, A 0.000, B 0.000, C 0.000 }
gfCNCPoint5[29944] = {X 73.9994, Y 14.6997, Z -8.0000, A 0.000, B 0.000, C 0.000 }
gfCNCPoint5[29945] = {X 73.9468, Y 15.0933, Z -8.0000, A 0.000, B 0.000, C 0.000 }
gfCNCPoint5[29946] = {X 77.7416, Y 25.2445, Z -8.0000, A 0.000, B 0.000, C 0.000 }
gfCNCPoint5[29947] = {X 80.1416, Y 25.2445, Z -8.0000, A 0.000, B 0.000, C 0.000 }
gfCNCPoint5[29948] = {X 80.1417, Y 17.4386, Z -8.0000, A 0.000, B 0.000, C 0.000 }
gfCNCPoint5[29949] = {X 79.4938, Y 16.4453, Z -8.0000, A 0.000, B 0.000, C 0.000 }
gfCNCPoint5[29950] = {X 79.0158, Y 15.3599, Z -8.0000, A 0.000, B 0.000, C 0.000 }
gfCNCPoint5[29951] = {X 78.7203, Y 14.2114, Z -8.0000, A 0.000, B 0.000, C 0.000 }
gfCNCPoint5[29952] = {X 78.6153, Y 13.0301, Z -8.0000, A 0.000, B 0.000, C 0.000 }
gfCNCPoint5[29953] = {X 78.6151, Y 12.1868, Z -8.0000, A 0.000, B 0.000, C 0.000 }
gfCNCPoint5[29954] = {X 78.6164, Y 12.0458, Z -8.0000, A 0.000, B 0.000, C 0.000 }
gfCNCPoint5[29955] = {X 78.6205, Y 11.9048, Z -8.0000, A 0.000, B 0.000, C 0.000 }
gfCNCPoint5[29956] = {X 71.6988, Y 11.9048, Z -8.0000, A 0.000, B 0.000, C 0.000 }
